(* Logix 5000 project; controller Proyecto_Final vendor 1 type 14 code 15 rev 16.42; software revision 16.03 *)

TASK MainTask (continuous, watchdog 500 ms) : MainProgram

MODULES
   Local : vendor 1 type 14 code 15 (SoftLogixController 2, rev 16.42)
END_MODULES

ADD_ON_INSTRUCTION Motorr   (* revision 1.0 *)
// Add On Motor
VAR_INPUT
   Cmd_Run : BOOL; {visible}   // Comando para acticar el motor en modo automatico
   Cmd_Stop : BOOL; {visible}   // Comando para detener el motor en modo automatico
   HMI_Run : BOOL;   // Comando para acticar el motor en modo manual
   HMI_Stop : BOOL;   // Comando para detener el motor en modo automatico
   Inp_Running : BOOL; {visible}   // Confirmacion de Falla del Motor
END_VAR
VAR_OUTPUT
   Sts_Running : BOOL; {visible}   // Estado activo del motor(salida fisica del PLC)
   Sts_RunFault : BOOL; {visible}   // Estado de falla del motor
END_VAR
VAR_INPUT
   Modo_Operacion : BOOL;
END_VAR
VAR
   Auto_Running : BOOL;
   Manu_Runnung : BOOL;
   TimerFault : TIMER := (PRE := 6000);
END_VAR

ROUTINE Logic   (* ladder *)
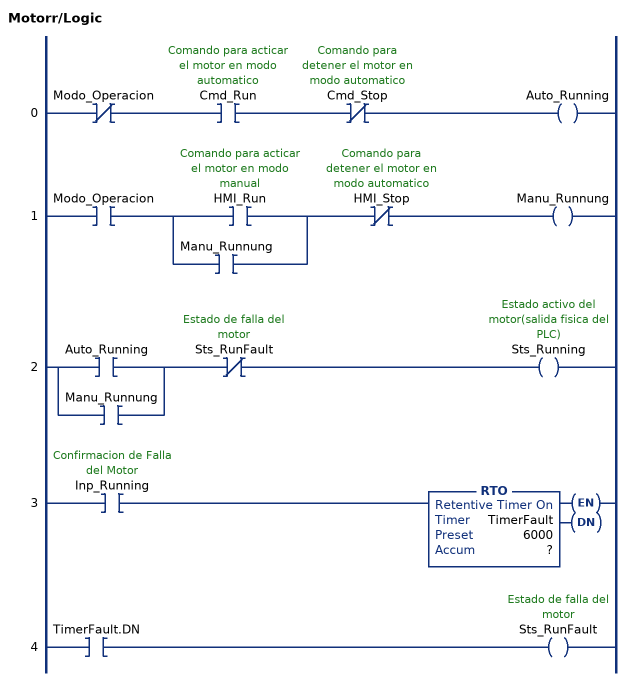
   0: XIO(Modo_Operacion)XIC(Cmd_Run)XIO(Cmd_Stop)OTE(Auto_Running);
   1: XIC(Modo_Operacion)[XIC(HMI_Run) ,XIC(Manu_Runnung) ]XIO(HMI_Stop)OTE(Manu_Runnung);
   2: [XIC(Auto_Running) ,XIC(Manu_Runnung) ]XIO(Sts_RunFault)OTE(Sts_Running);
   3: XIC(Inp_Running)RTO(TimerFault,?,?);
   4: XIC(TimerFault.DN)OTE(Sts_RunFault);
END_ROUTINE
END_ADD_ON_INSTRUCTION

ADD_ON_INSTRUCTION PICK_AND_PLACE   (* revision 1.0 *)
VAR_OUTPUT
   Banda_Entry_Conveyor : BOOL; {visible}
   Move_z : BOOL; {visible}
   Grab : BOOL; {visible}
   Move_x : BOOL; {visible}
   Banda_Exit_Conveyor : BOOL; {visible}
END_VAR
VAR_INPUT
   Sensor_Item_at_entry : BOOL;
   Sensor_Item_detected : BOOL;
   Sensor_Item_at_exit : BOOL;
   Cmd_Run_Banda_Entry_Conveyor : BOOL; {visible}
   Cmd_Run_Move_z : BOOL; {visible}
   Cmd_Run_Grab : BOOL; {visible}
   Cmd_Run_Move_x : BOOL; {visible}
   Cmd_Run_Banda_Exit_Conveyor : BOOL; {visible}
   Modo_Operacion : BOOL;
   Sensor_Entry : BOOL;
END_VAR

ROUTINE Logic   (* ladder *)
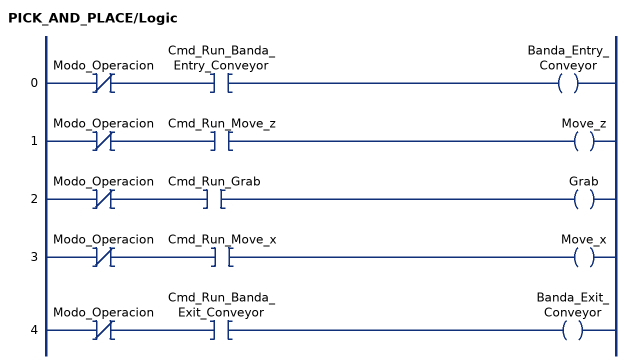
   0: XIO(Modo_Operacion)XIC(Cmd_Run_Banda_Entry_Conveyor)OTE(Banda_Entry_Conveyor);
   1: XIO(Modo_Operacion)XIC(Cmd_Run_Move_z)OTE(Move_z);
   2: XIO(Modo_Operacion)XIC(Cmd_Run_Grab)OTE(Grab);
   3: XIO(Modo_Operacion)XIC(Cmd_Run_Move_x)OTE(Move_x);
   4: XIO(Modo_Operacion)XIC(Cmd_Run_Banda_Exit_Conveyor)OTE(Banda_Exit_Conveyor);
END_ROUTINE
END_ADD_ON_INSTRUCTION

ADD_ON_INSTRUCTION PICK_AND_PLACE_XYZ   (* revision 1.0 *)
VAR_INPUT
   Modo_Operacion : BOOL; {visible}
   Cmd_Run_Pallet_Conveyor : BOOL; {visible}
   Cmd_Run_Part_Conveyor : BOOL; {visible}
   Cmd_Run_GradXYZ : BOOL; {visible}
END_VAR
VAR_OUTPUT
   Pallet_Conveyor : BOOL; {visible}
   Part_Conveyor : BOOL; {visible}
END_VAR
VAR_INPUT
   Sensor_Pallet : BOOL;
   Sensor_Part : BOOL;
   Sensor_Deteccion : BOOL;
END_VAR
VAR_OUTPUT
   V_Eje_X : REAL; {visible}
   V_Eje_Y : REAL; {visible}
   V_Eje_Z : REAL; {visible}
   GradXYZ : BOOL;
END_VAR
VAR_INPUT
   Sensor_Entry : BOOL;
   Cmd_Run_Emiter_Pallets : BOOL; {visible}
END_VAR
VAR_OUTPUT
   Emiter_Pallets : BOOL; {visible}
END_VAR

ROUTINE Logic   (* ladder *)
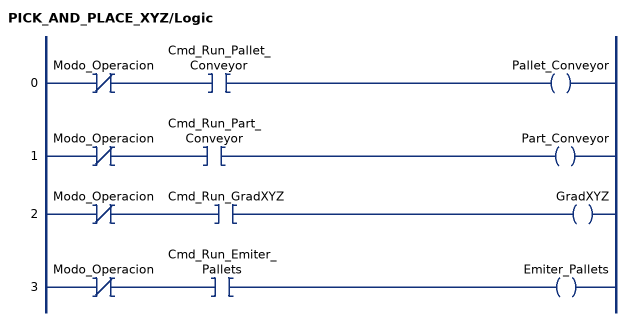
   0: XIO(Modo_Operacion)XIC(Cmd_Run_Pallet_Conveyor)OTE(Pallet_Conveyor);
   1: XIO(Modo_Operacion)XIC(Cmd_Run_Part_Conveyor)OTE(Part_Conveyor);
   2: XIO(Modo_Operacion)XIC(Cmd_Run_GradXYZ)OTE(GradXYZ);
   3: XIO(Modo_Operacion)XIC(Cmd_Run_Emiter_Pallets)OTE(Emiter_Pallets);
END_ROUTINE
END_ADD_ON_INSTRUCTION

ADD_ON_INSTRUCTION PRODUCTION_LINE   (* revision 1.0 *)
VAR_INPUT
   Modo_Operacion : BOOL; {visible}
   Cmd_Run_Banda_Lids_In : BOOL; {visible}
   Cmd_Run_Brazo : BOOL; {visible}
   Cmd_Run_Banda_Lids_Out1 : BOOL; {visible}
   Cmd_Run_Banda_Lids_Out2 : BOOL; {visible}
END_VAR
VAR_OUTPUT
   Banda_Lids_In : BOOL; {visible}
   Banda_Lids_Out1 : BOOL; {visible}
   Banda_Lids_Out2 : BOOL; {visible}
END_VAR
VAR_INPUT
   Sensor_Lid_In : BOOL;
   Sensor_Lid_Out : BOOL;
END_VAR
VAR_OUTPUT
   Brazo : BOOL; {visible}
END_VAR

ROUTINE Logic   (* ladder *)
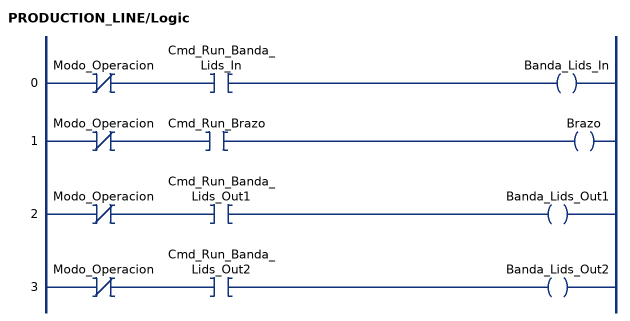
   0: XIO(Modo_Operacion)XIC(Cmd_Run_Banda_Lids_In)OTE(Banda_Lids_In);
   1: XIO(Modo_Operacion)XIC(Cmd_Run_Brazo)OTE(Brazo);
   2: XIO(Modo_Operacion)XIC(Cmd_Run_Banda_Lids_Out1)OTE(Banda_Lids_Out1);
   3: XIO(Modo_Operacion)XIC(Cmd_Run_Banda_Lids_Out2)OTE(Banda_Lids_Out2);
END_ROUTINE
END_ADD_ON_INSTRUCTION

ADD_ON_INSTRUCTION SCENE_1   (* revision 1.0 *)
VAR_INPUT
   Modo_Operacion : BOOL;   // Comando para cambiar el Modo_Automatico_Manual
   Item_at_entry : BOOL; {visible}
   Item_detected : BOOL; {visible}
   Item_at_exit : BOOL; {visible}
END_VAR
VAR_OUTPUT
   Entry_conveyor : BOOL; {visible}
   Move_z : BOOL; {visible}
   Grab : BOOL; {visible}
   Move_x : BOOL; {visible}
   Exit_coneyor : BOOL; {visible}
END_VAR
VAR_INPUT
   Incio : BOOL; {visible}
   Mover_Banda_1 : BOOL; {visible}
END_VAR
VAR_OUTPUT
   Banda_1 : BOOL; {visible}
END_VAR
VAR_INPUT
   Mover_eje_z : BOOL; {visible}
   Sostener_Pieza : BOOL; {visible}
   Mover_banda_2 : BOOL; {visible}
   Mover_eje_x : BOOL; {visible}
END_VAR
VAR
   Timer_Axis : TIMER := (PRE := 1000);
   Inicio : BOOL;
END_VAR

ROUTINE Logic   (* ladder *)
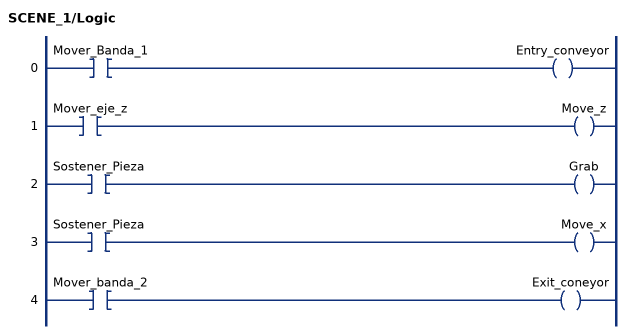
   0: XIC(Mover_Banda_1)OTE(Entry_conveyor);
   1: XIC(Mover_eje_z)OTE(Move_z);
   2: XIC(Sostener_Pieza)OTE(Grab);
   3: XIC(Sostener_Pieza)OTE(Move_x);
   4: XIC(Mover_banda_2)OTE(Exit_coneyor);
END_ROUTINE
END_ADD_ON_INSTRUCTION

ADD_ON_INSTRUCTION SEPARATION_STATION   (* revision 1.0 *)
VAR_INPUT
   Modo_Operacion : BOOL; {visible}
   Cmd_Run_Banda_Conveyor : BOOL; {visible}
   Cmd_Run_Pusher_Green : BOOL; {visible}
   Cmd_Run_Pusher_Blue : BOOL; {visible}
   Sensor_Piezas_Green : DINT; {visible}
   Sensor_Piezas_Blue : DINT; {visible}
END_VAR
VAR_OUTPUT
   Banda_Conveyor : BOOL; {visible}
   Pusher_Green : BOOL; {visible}
   Pusher_Bluee : BOOL; {visible}
END_VAR
VAR_INPUT
   Sensor_Entry : BOOL;
END_VAR

ROUTINE Logic   (* ladder *)
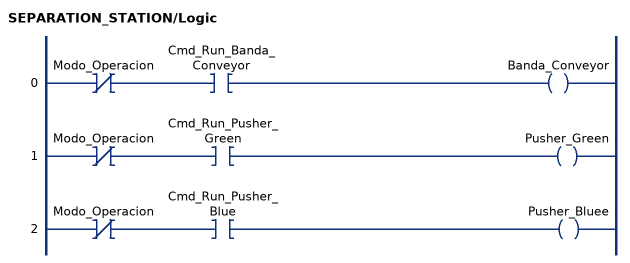
   0: XIO(Modo_Operacion)XIC(Cmd_Run_Banda_Conveyor)OTE(Banda_Conveyor);
   1: XIO(Modo_Operacion)XIC(Cmd_Run_Pusher_Green)OTE(Pusher_Green);
   2: XIO(Modo_Operacion)XIC(Cmd_Run_Pusher_Blue)OTE(Pusher_Bluee);
END_ROUTINE
END_ADD_ON_INSTRUCTION

ADD_ON_INSTRUCTION SORTING_BY_HEIGHT   (* revision 1.0 *)
VAR_INPUT
   Modo_Operacion : BOOL; {visible}
   Cmd_Run_Conveyor_Entry : BOOL; {visible}
   Cmd_Run_Load : BOOL; {visible}
   Cmd_Run_Turn : BOOL; {visible}
   Cmd_Run_Conveyor_Right : BOOL; {visible}
   Cmd_Run_Conveyor_Left : BOOL; {visible}
   Cmd_Run_Un_Load : BOOL; {visible}
END_VAR
VAR_OUTPUT
   Conveyor_Entry : BOOL; {visible}
   Load : BOOL; {visible}
   Turn : BOOL; {visible}
   Conveyor_Right : BOOL; {visible}
   Conveyor_Left : BOOL; {visible}
   Un_Load : BOOL; {visible}
END_VAR
VAR_INPUT
   Sensor_Low : BOOL;
   Sensor_High : BOOL;
   Sensor_Final_Conveyor_Entry : BOOL;
   Sensor_Front : BOOL;
   Sensor_In_Right_Conveyor : BOOL;
   Sensor_In_Left_Conveyor : BOOL;
   Sensor_Entry : BOOL;
END_VAR

ROUTINE Logic   (* ladder *)
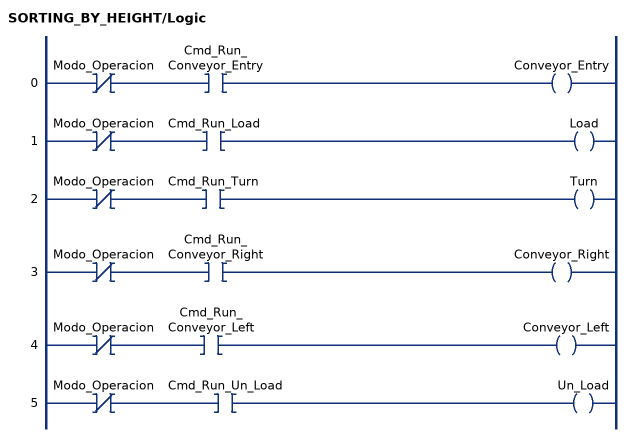
   0: XIO(Modo_Operacion)XIC(Cmd_Run_Conveyor_Entry)OTE(Conveyor_Entry);
   1: XIO(Modo_Operacion)XIC(Cmd_Run_Load)OTE(Load);
   2: XIO(Modo_Operacion)XIC(Cmd_Run_Turn)OTE(Turn);
   3: XIO(Modo_Operacion)XIC(Cmd_Run_Conveyor_Right)OTE(Conveyor_Right);
   4: XIO(Modo_Operacion)XIC(Cmd_Run_Conveyor_Left)OTE(Conveyor_Left);
   5: XIO(Modo_Operacion)XIC(Cmd_Run_Un_Load)OTE(Un_Load);
END_ROUTINE
END_ADD_ON_INSTRUCTION

ADD_ON_INSTRUCTION SORTING_BY_WEIGHT   (* revision 1.0 *)
VAR_INPUT
   Modo_Operacion : BOOL; {visible}
   Cmd_Run_Conveyor_Entry : BOOL; {visible}
   Cmd_Run_Conveyor_Peso : BOOL; {visible}
   Cmd_Run_Send_Adelante : BOOL; {visible}
   Cmd_Run_Send_Right : BOOL; {visible}
   Cmd_Run_Send_Left : BOOL; {visible}
   Cmd_Run_Conveyor_Right : BOOL; {visible}
   Cmd_Run_Conveyor_Left : BOOL; {visible}
   Cmd_Run_Conveyor_Front : BOOL; {visible}
END_VAR
VAR_OUTPUT
   Conveyor_Entry : BOOL; {visible}
   Conveyor_Peso : BOOL; {visible}
   Send_Adelante : BOOL; {visible}
   Send_Right : BOOL; {visible}
   Send_Left : BOOL; {visible}
   Conveyor_Right : BOOL; {visible}
   Conveyor_Left : BOOL; {visible}
   Conveyor_Front : BOOL; {visible}
END_VAR
VAR_INPUT
   Sensor_Peso : REAL; {visible}
   Sensor_Conveyor_Entry : BOOL;
   Sensor_Conveyor_In_Right : BOOL;
   Sensor_Conveyor_In_Left : BOOL;
   Sensor_Conveyor_In_Front : BOOL;
END_VAR

ROUTINE Logic   (* ladder *)
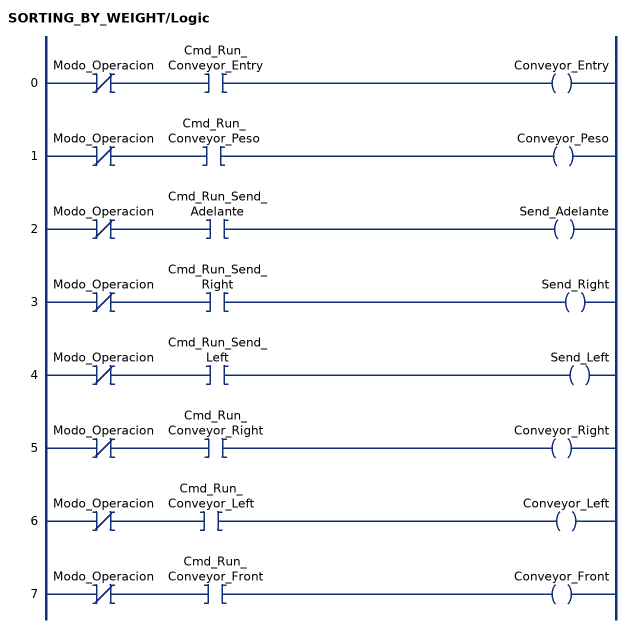
   0: XIO(Modo_Operacion)XIC(Cmd_Run_Conveyor_Entry)OTE(Conveyor_Entry);
   1: XIO(Modo_Operacion)XIC(Cmd_Run_Conveyor_Peso)OTE(Conveyor_Peso);
   2: XIO(Modo_Operacion)XIC(Cmd_Run_Send_Adelante)OTE(Send_Adelante);
   3: XIO(Modo_Operacion)XIC(Cmd_Run_Send_Right)OTE(Send_Right);
   4: XIO(Modo_Operacion)XIC(Cmd_Run_Send_Left)OTE(Send_Left);
   5: XIO(Modo_Operacion)XIC(Cmd_Run_Conveyor_Right)OTE(Conveyor_Right);
   6: XIO(Modo_Operacion)XIC(Cmd_Run_Conveyor_Left)OTE(Conveyor_Left);
   7: XIO(Modo_Operacion)XIC(Cmd_Run_Conveyor_Front)OTE(Conveyor_Front);
END_ROUTINE
END_ADD_ON_INSTRUCTION

VAR_GLOBAL   (* controller tags *)
   A1 : SFC_STEP;
   AAAA : SFC_STEP;
   Altura : SORTING_BY_HEIGHT;
   AZU : BOOL;
   B1 : SFC_STEP;
   BBB : SFC_STEP;
   BBB_001 : SFC_STEP;
   BBB_002 : SFC_STEP;
   BBB_003 : SFC_STEP;
   BOOL_IN_0 : ALIAS FOR Proceso.Sensor_Item_at_entry;
   BOOL_IN_1 : ALIAS FOR Proceso.Sensor_Item_detected;
   BOOL_IN_10 : ALIAS FOR Proceso2.Sensor_Entry;
   BOOL_IN_11 : ALIAS FOR STARTR;
   BOOL_IN_12 : ALIAS FOR Linea1.Sensor_Lid_In;
   BOOL_IN_13 : ALIAS FOR Linea1.Sensor_Lid_Out;
   BOOL_IN_14 : ALIAS FOR Linea2.Sensor_Lid_In;
   BOOL_IN_15 : ALIAS FOR Linea2.Sensor_Lid_Out;
   BOOL_IN_16 : ALIAS FOR Proceso.Sensor_Entry;
   BOOL_IN_17 : ALIAS FOR XYZ.Sensor_Pallet;
   BOOL_IN_18 : ALIAS FOR XYZ.Sensor_Part;
   BOOL_IN_19 : ALIAS FOR XYZ.Sensor_Deteccion;
   BOOL_IN_2 : ALIAS FOR Proceso.Sensor_Item_at_exit;
   BOOL_IN_20 : ALIAS FOR SEPARA.Sensor_Entry;
   BOOL_IN_21 : ALIAS FOR Altura.Sensor_Low;
   BOOL_IN_22 : ALIAS FOR Altura.Sensor_Final_Conveyor_Entry;
   BOOL_IN_23 : ALIAS FOR Altura.Sensor_Front;
   BOOL_IN_24 : ALIAS FOR Altura.Sensor_In_Right_Conveyor;
   BOOL_IN_25 : ALIAS FOR Altura.Sensor_High;
   BOOL_IN_26 : ALIAS FOR Altura.Sensor_In_Left_Conveyor;
   BOOL_IN_27 : ALIAS FOR Peso.Sensor_Conveyor_Entry;
   BOOL_IN_28 : ALIAS FOR Peso.Sensor_Conveyor_In_Right;
   BOOL_IN_29 : ALIAS FOR Peso.Sensor_Conveyor_In_Left;
   BOOL_IN_3 : ALIAS FOR Line3.Sensor_Lid_In;
   BOOL_IN_30 : ALIAS FOR Peso.Sensor_Conveyor_In_Front;
   BOOL_IN_31 : ALIAS FOR REARME;
   BOOL_IN_32 : ALIAS FOR STOPSITO;
   BOOL_IN_4 : ALIAS FOR Line3.Sensor_Lid_Out;
   BOOL_IN_5 : ALIAS FOR XYZ.Sensor_Entry;
   BOOL_IN_6 : ALIAS FOR Altura.Sensor_Entry;
   BOOL_IN_7 : ALIAS FOR Proceso2.Sensor_Item_at_entry;
   BOOL_IN_8 : ALIAS FOR Proceso2.Sensor_Item_detected;
   BOOL_IN_9 : ALIAS FOR Proceso2.Sensor_Item_at_exit;
   BOOL_OUT_0 : ALIAS FOR Proceso.Banda_Entry_Conveyor;
   BOOL_OUT_1 : ALIAS FOR Proceso.Move_z;
   BOOL_OUT_10 : ALIAS FOR Line3.Banda_Lids_Out1;
   BOOL_OUT_11 : ALIAS FOR Line3.Banda_Lids_Out2;
   BOOL_OUT_12 : ALIAS FOR Linea1.Banda_Lids_In;
   BOOL_OUT_13 : ALIAS FOR Linea1.Brazo;
   BOOL_OUT_14 : ALIAS FOR Linea1.Banda_Lids_Out1;
   BOOL_OUT_15 : ALIAS FOR Linea1.Banda_Lids_Out2;
   BOOL_OUT_16 : ALIAS FOR Linea2.Banda_Lids_In;
   BOOL_OUT_17 : ALIAS FOR Linea2.Brazo;
   BOOL_OUT_18 : ALIAS FOR Linea2.Banda_Lids_Out1;
   BOOL_OUT_19 : ALIAS FOR Linea2.Banda_Lids_Out2;
   BOOL_OUT_2 : ALIAS FOR Proceso.Grab;
   BOOL_OUT_20 : ALIAS FOR XYZ.Pallet_Conveyor;
   BOOL_OUT_21 : ALIAS FOR XYZ.Part_Conveyor;
   BOOL_OUT_22 : ALIAS FOR XYZ.GradXYZ;
   BOOL_OUT_23 : ALIAS FOR Altura.Conveyor_Entry;
   BOOL_OUT_24 : ALIAS FOR Altura.Load;
   BOOL_OUT_25 : ALIAS FOR Altura.Turn;
   BOOL_OUT_26 : ALIAS FOR Altura.Conveyor_Right;
   BOOL_OUT_27 : ALIAS FOR Altura.Un_Load;
   BOOL_OUT_28 : ALIAS FOR Altura.Conveyor_Left;
   BOOL_OUT_29 : ALIAS FOR Peso.Conveyor_Entry;
   BOOL_OUT_3 : ALIAS FOR Proceso.Move_x;
   BOOL_OUT_30 : ALIAS FOR Peso.Conveyor_Peso;
   BOOL_OUT_31 : ALIAS FOR Peso.Send_Right;
   BOOL_OUT_32 : ALIAS FOR Peso.Send_Adelante;
   BOOL_OUT_33 : ALIAS FOR Peso.Conveyor_Right;
   BOOL_OUT_34 : ALIAS FOR Peso.Send_Left;
   BOOL_OUT_35 : ALIAS FOR Peso.Conveyor_Left;
   BOOL_OUT_36 : ALIAS FOR Peso.Conveyor_Front;
   BOOL_OUT_37 : ALIAS FOR XYZ.Emiter_Pallets;
   BOOL_OUT_39 : ALIAS FOR Proceso2.Move_z;
   BOOL_OUT_4 : ALIAS FOR Proceso.Banda_Exit_Conveyor;
   BOOL_OUT_40 : ALIAS FOR Proceso2.Grab;
   BOOL_OUT_41 : ALIAS FOR Proceso2.Move_x;
   BOOL_OUT_42 : ALIAS FOR Proceso2.Banda_Entry_Conveyor;
   BOOL_OUT_43 : ALIAS FOR Proceso2.Banda_Exit_Conveyor;
   BOOL_OUT_5 : ALIAS FOR SEPARA.Banda_Conveyor;
   BOOL_OUT_6 : ALIAS FOR SEPARA.Pusher_Green;
   BOOL_OUT_7 : ALIAS FOR SEPARA.Pusher_Bluee;
   BOOL_OUT_8 : ALIAS FOR Line3.Banda_Lids_In;
   BOOL_OUT_9 : ALIAS FOR Line3.Brazo;
   C1 : SFC_STEP;
   CC : SFC_STEP;
   CC_001 : SFC_STEP;
   CC_002 : SFC_STEP;
   CC_003 : SFC_STEP;
   CMD_1 : BOOL;
   CMD_2 : BOOL;
   CMD_3 : BOOL;
   Cmd_banda1 : BOOL;
   Cmd_banda2 : BOOL;
   Cmd_banda3 : BOOL;
   CMD_banda_derecha : BOOL;
   CMD_banda_Front : BOOL;
   CMD_banda_IZQQ : BOOL;
   Cmd_bandaCLAS : BOOL;
   CMD_conveyor_entry : BOOL;
   CMD_conveyor_peso : BOOL;
   CMD_DETEC : BOOL;
   Cmd_giro : BOOL;
   CMD_LEFT : BOOL;
   Cmd_LOAD : BOOL;
   CMD_RIFHT : BOOL;
   CMD_Send_Front : BOOL;
   CMD_Send_LEFT : BOOL;
   CMD_Send_righ : BOOL;
   CMD_Send_ruedas : BOOL;
   Cmd_Turn : BOOL;
   CMD_UNLOAD : BOOL;
   CMD_X : BOOL;
   CMD_X0 : BOOL;
   CMD_X2 : BOOL;
   CMD_Y : BOOL;
   CMD_Y0 : BOOL;
   CMD_Y2 : BOOL;
   CMD_Z : BOOL;
   CMD_Z0 : BOOL;
   CMD_Z2 : BOOL;
   CMDGIRO : BOOL;
   D1 : SFC_STEP;
   DD : SFC_STEP;
   DD_001 : SFC_STEP;
   DD_002 : SFC_STEP;
   DD_003 : SFC_STEP;
   DF : SFC_STEP := (PRE := 100);
   DF_001 : SFC_STEP := (PRE := 100);
   DF_002 : SFC_STEP := (PRE := 100);
   DFR : SFC_STEP := (PRE := 4000);
   E1 : SFC_STEP := (PRE := 2500);
   E1_001 : SFC_STEP := (PRE := 2500);
   E1_002 : SFC_STEP := (PRE := 2500);
   E2 : SFC_STEP;
   E2_001 : SFC_STEP;
   E2_002 : SFC_STEP;
   E3 : SFC_STEP := (PRE := 1200);
   E3_001 : SFC_STEP := (PRE := 1200);
   E3_002 : SFC_STEP := (PRE := 1200);
   E3_003 : SFC_STEP := (PRE := 1200);
   E3_004 : SFC_STEP := (PRE := 1200);
   E3_005 : SFC_STEP := (PRE := 1200);
   E3_006 : SFC_STEP := (PRE := 1200);
   E3_007 : SFC_STEP := (PRE := 1200);
   E4 : SFC_STEP := (PRE := 600);
   E4_001 : SFC_STEP := (PRE := 600);
   E4_002 : SFC_STEP := (PRE := 600);
   E4_003 : SFC_STEP := (PRE := 425);
   E4_004 : SFC_STEP := (PRE := 600);
   E4_005 : SFC_STEP := (PRE := 425);
   E4_006 : SFC_STEP := (PRE := 350);
   E4_007 : SFC_STEP := (PRE := 600);
   EE : SFC_STEP := (PRE := 350);
   EE_001 : SFC_STEP := (PRE := 350);
   EE_002 : SFC_STEP := (PRE := 350);
   EE_003 : SFC_STEP := (PRE := 350);
   EO : DINT;
   EOwww : SFC_STEP;
   EOwww_001 : SFC_STEP;
   ERT : SFC_STEP;
   ERTT : SFC_STEP;
   ERTT_001 : SFC_STEP;
   ERTT_002 : SFC_STEP;
   ET1 : SFC_STEP;
   ET10 : SFC_STEP := (PRE := 1200);
   ET11 : SFC_STEP := (PRE := 1200);
   ET12 : SFC_STEP;
   ET122 : SFC_STEP;
   ET3 : SFC_STEP;
   ET4 : SFC_STEP;
   ET4_001 : SFC_STEP;
   ET5 : SFC_STEP;
   ET5_001 : SFC_STEP;
   ET6 : SFC_STEP;
   ET7 : SFC_STEP;
   ET8 : SFC_STEP;
   ET89 : SFC_STEP;
   ET9 : SFC_STEP := (PRE := 1200);
   ETP1 : SFC_STEP;
   ETP2 : SFC_STEP;
   ETP22 : SFC_STEP := (PRE := 2500);
   ETP3 : SFC_STEP;
   ETP4 : SFC_STEP := (PRE := 1200);
   ETP5 : SFC_STEP := (PRE := 600);
   ETP6 : SFC_STEP := (PRE := 4000);
   ETP66 : SFC_STEP := (PRE := 2700);
   ETY1 : SFC_STEP := (PRE := 4000);
   ETY1_001 : SFC_STEP := (PRE := 4000);
   EYT : SFC_STEP;
   F1 : SFC_STEP := (PRE := 3000);
   F1_001 : SFC_STEP := (PRE := 3000);
   FF : SFC_STEP := (PRE := 1000);
   FF_001 : SFC_STEP := (PRE := 1000);
   FF_002 : SFC_STEP := (PRE := 1000);
   FF_003 : SFC_STEP := (PRE := 1000);
   FG : SFC_STEP;
   FG_001 : SFC_STEP;
   FG_002 : SFC_STEP;
   FLOAT_IN_0 : REAL;
   FLOAT_IN_1 : DINT;
   FLOAT_IN_2 : REAL;
   FLOAT_IN_3 : ALIAS FOR Peso.Sensor_Peso;
   FLOAT_IN_ON : DINT;
   FLOAT_OUT_0 : ALIAS FOR XYZ.V_Eje_X;
   FLOAT_OUT_1 : ALIAS FOR XYZ.V_Eje_Y;
   FLOAT_OUT_2 : ALIAS FOR XYZ.V_Eje_Z;
   G1 : SFC_STEP;
   GGG : SFC_STEP := (PRE := 150);
   GGG_001 : SFC_STEP := (PRE := 150);
   GGG_002 : SFC_STEP := (PRE := 150);
   GGG_003 : SFC_STEP := (PRE := 150);
   III : SFC_STEP;
   INT_IN_0 : ALIAS FOR SEPARA.Sensor_Piezas_Blue;
   INT_IN_1 : ALIAS FOR SEPARA.Sensor_Piezas_Green;
   INT_OUT_0 : REAL;
   INT_OUT_1 : DINT;
   INT_OUT_O : DINT;
   IO : SFC_STEP;
   IO_001 : SFC_STEP;
   IO_002 : SFC_STEP;
   KKK : SFC_STEP := (PRE := 7000);
   KKK_001 : SFC_STEP := (PRE := 4000);
   Line3 : PRODUCTION_LINE;
   Linea1 : PRODUCTION_LINE;
   Linea2 : PRODUCTION_LINE;
   Modo_Operacion : BOOL;
   Peso : SORTING_BY_WEIGHT;
   Proceso : PICK_AND_PLACE;
   Proceso1 : BOOL;
   Proceso2 : PICK_AND_PLACE;
   prueba : TIMER := (PRE := 6);
   QW : SFC_STEP;
   RE : SFC_STEP := (PRE := 330);
   RE_001 : SFC_STEP := (PRE := 330);
   RE_002 : SFC_STEP := (PRE := 330);
   REARME : BOOL;
   REPIT : SFC_STEP;
   RRR : SFC_STEP;
   RRR_001 : SFC_STEP;
   RRR_002 : SFC_STEP;
   RT : SFC_STEP;
   RT_001 : SFC_STEP;
   RT_002 : SFC_STEP;
   SEPARA : SEPARATION_STATION;
   START1 : BOOL;
   STARTR : BOOL;
   STARTT : BOOL;
   STOP2 : BOOL;
   STOPSITO : BOOL;
   SYS_0N : BOOL;
   T2 : SFC_STEP;
   T2_001 : SFC_STEP;
   T2_002 : SFC_STEP;
   test : BOOL;
   TESTTT : TIMER := (PRE := 6);
   testttt : TIMER := (PRE := 5000);
   tiempo : BOOL;
   TR : SFC_STEP;
   TR_001 : SFC_STEP;
   TR_002 : SFC_STEP;
   TTT : BOOL;
   ty : SFC_STEP := (Count := 2);
   V1 : SFC_STEP := (PRE := 3000);
   VER : BOOL;
   WE : SFC_STEP;
   WEE : SFC_STEP := (PRE := 1000);
   WEE_001 : SFC_STEP := (PRE := 1000);
   WERR : SFC_STEP;
   X1 : SFC_STEP;
   XX : SFC_STEP;
   XX_001 : SFC_STEP;
   XX_002 : SFC_STEP;
   XYZ : PICK_AND_PLACE_XYZ;
   Y1 : SFC_STEP := (PRE := 2500);
   Z1 : SFC_STEP;
END_VAR

PROGRAM MainProgram   (* main routine MainRoutine *)
VAR
   Action_000 : SFC_ACTION;
   Action_001 : SFC_ACTION;
   Action_002 : SFC_ACTION;
   Action_003 : SFC_ACTION;
   Action_004 : SFC_ACTION;
   Action_005 : SFC_ACTION;
   Action_006 : SFC_ACTION;
   Action_007 : SFC_ACTION;
   Action_008 : SFC_ACTION;
   Action_009 : SFC_ACTION;
   Action_010 : SFC_ACTION;
   Action_011 : SFC_ACTION;
   Action_012 : SFC_ACTION;
   Action_013 : SFC_ACTION;
   Action_014 : SFC_ACTION;
   Action_015 : SFC_ACTION;
   Action_016 : SFC_ACTION;
   Action_017 : SFC_ACTION;
   Action_018 : SFC_ACTION;
   Action_019 : SFC_ACTION;
   Action_020 : SFC_ACTION;
   Action_021 : SFC_ACTION;
   Action_022 : SFC_ACTION;
   Action_023 : SFC_ACTION;
   Action_024 : SFC_ACTION;
   Action_025 : SFC_ACTION;
   Action_026 : SFC_ACTION;
   Action_027 : SFC_ACTION;
   Action_028 : SFC_ACTION;
   Action_029 : SFC_ACTION;
   Action_030 : SFC_ACTION;
   Action_031 : SFC_ACTION;
   Action_032 : SFC_ACTION;
   Action_033 : SFC_ACTION;
   Action_034 : SFC_ACTION;
   Action_035 : SFC_ACTION;
   Action_036 : SFC_ACTION;
   Action_037 : SFC_ACTION;
   Action_038 : SFC_ACTION;
   Action_039 : SFC_ACTION;
   Action_040 : SFC_ACTION;
   Action_041 : SFC_ACTION;
   Action_042 : SFC_ACTION;
   Action_043 : SFC_ACTION;
   Action_044 : SFC_ACTION;
   Action_045 : SFC_ACTION;
   Action_046 : SFC_ACTION;
   Action_047 : SFC_ACTION;
   Action_048 : SFC_ACTION;
   Action_049 : SFC_ACTION;
   Action_050 : SFC_ACTION;
   Action_051 : SFC_ACTION;
   Action_052 : SFC_ACTION;
   Action_053 : SFC_ACTION;
   Action_054 : SFC_ACTION;
   Action_055 : SFC_ACTION;
   Action_056 : SFC_ACTION;
   Action_057 : SFC_ACTION;
   Action_058 : SFC_ACTION;
   Action_059 : SFC_ACTION;
   Action_060 : SFC_ACTION;
   Action_061 : SFC_ACTION;
   Action_062 : SFC_ACTION;
   Action_063 : SFC_ACTION;
   Action_064 : SFC_ACTION;
   Action_065 : SFC_ACTION;
   Action_066 : SFC_ACTION;
   Action_067 : SFC_ACTION;
   Action_068 : SFC_ACTION;
   Action_069 : SFC_ACTION;
   Action_070 : SFC_ACTION;
   Action_071 : SFC_ACTION;
   Action_072 : SFC_ACTION;
   Action_073 : SFC_ACTION;
   Action_074 : SFC_ACTION;
   Action_075 : SFC_ACTION;
   Action_076 : SFC_ACTION;
   Action_077 : SFC_ACTION;
   Action_078 : SFC_ACTION;
   Action_079 : SFC_ACTION;
   Action_080 : SFC_ACTION;
   Action_081 : SFC_ACTION;
   Action_082 : SFC_ACTION;
   Action_083 : SFC_ACTION;
   Action_084 : SFC_ACTION;
   Action_085 : SFC_ACTION;
   Action_086 : SFC_ACTION;
   Action_087 : SFC_ACTION;
   Action_088 : SFC_ACTION;
   Action_089 : SFC_ACTION;
   Action_090 : SFC_ACTION;
   Action_091 : SFC_ACTION;
   Action_092 : SFC_ACTION;
   Action_093 : SFC_ACTION;
   Action_094 : SFC_ACTION;
   Action_095 : SFC_ACTION;
   Action_096 : SFC_ACTION;
   Action_097 : SFC_ACTION;
   Action_098 : SFC_ACTION;
   ESCENA_1_01 : PICK_AND_PLACE;
   HIGH : DINT;
   Linea3 : PRODUCTION_LINE;
   Motorr_01 : Motorr;
   PICK_AND_PLACE_01 : PICK_AND_PLACE;
   PICK_AND_PLACE_XYZ_01 : PICK_AND_PLACE_XYZ;
   PRODUCTION_LINE_01 : PRODUCTION_LINE;
   SCENE_1_01 : SCENE_1;
   SEPARATIN_STATION_01 : SEPARATION_STATION;
   SORTING_BY_HEIGHT_01 : SORTING_BY_HEIGHT;
   SORTING_BY_WEIGHT_01 : SORTING_BY_WEIGHT;
   Step_000 : SFC_STEP;
   Step_001 : SFC_STEP;
   Step_002 : SFC_STEP;
   Step_003 : SFC_STEP;
   Step_004 : SFC_STEP;
   Step_005 : SFC_STEP;
   Step_006 : SFC_STEP;
   Step_007 : SFC_STEP;
   Step_008 : SFC_STEP;
   Step_009 : SFC_STEP;
   Step_010 : SFC_STEP;
   Step_011 : SFC_STEP;
   Step_012 : SFC_STEP;
   Step_013 : SFC_STEP := (PRE := 850);
   Step_014 : SFC_STEP := (PRE := 1000);
   Step_015 : SFC_STEP := (PRE := 1000);
   Step_016 : SFC_STEP := (PRE := 850);
   Step_017 : SFC_STEP;
   Step_018 : SFC_STEP;
   Step_019 : SFC_STEP;
   Step_020 : SFC_STEP;
   Step_021 : SFC_STEP;
   Step_022 : SFC_STEP;
   Step_023 : SFC_STEP;
   Step_024 : SFC_STEP;
   Step_025 : SFC_STEP;
   Step_026 : SFC_STEP;
   Step_027 : SFC_STEP;
   Step_028 : SFC_STEP;
   Step_029 : SFC_STEP;
   Step_030 : SFC_STEP;
   Step_031 : SFC_STEP;
   Step_032 : SFC_STEP;
   Step_033 : SFC_STEP;
   Step_034 : SFC_STEP;
   Step_035 : SFC_STEP;
   Step_036 : SFC_STEP;
   Step_037 : SFC_STEP;
   Step_038 : SFC_STEP;
   Step_039 : SFC_STEP;
   Step_040 : SFC_STEP;
   Step_041 : SFC_STEP;
   Step_042 : SFC_STEP;
   Step_043 : SFC_STEP;
   Step_044 : SFC_STEP;
   Step_045 : SFC_STEP;
   Step_046 : SFC_STEP;
   Step_047 : SFC_STEP;
   Step_048 : SFC_STEP;
   Step_049 : SFC_STEP;
   Step_050 : SFC_STEP;
   Step_051 : SFC_STEP := (PRE := 5000);
   Step_052 : SFC_STEP;
   Step_053 : SFC_STEP;
   Step_054 : SFC_STEP;
   Step_055 : SFC_STEP;
   Step_056 : SFC_STEP;
   Step_057 : SFC_STEP;
   Step_058 : SFC_STEP;
   Step_059 : SFC_STEP;
   Step_060 : SFC_STEP;
   Step_061 : SFC_STEP;
   Step_062 : SFC_STEP;
   Step_063 : SFC_STEP;
   Step_064 : SFC_STEP := (PRE := 1200);
   Step_065 : SFC_STEP;
   Step_066 : SFC_STEP;
   Step_067 : SFC_STEP;
   Step_068 : SFC_STEP;
   Tran_000 : BOOL;
   Tran_001 : BOOL;
   Tran_002 : BOOL;
   Tran_003 : BOOL;
   Tran_004 : BOOL;
   Tran_005 : BOOL;
   Tran_006 : BOOL;
   Tran_007 : BOOL;
   Tran_008 : BOOL;
   Tran_009 : BOOL;
   Tran_010 : BOOL;
   Tran_011 : BOOL;
   Tran_012 : BOOL;
   Tran_013 : BOOL;
   Tran_014 : BOOL;
   Tran_015 : BOOL;
   Tran_016 : BOOL;
   Tran_017 : BOOL;
   Tran_018 : BOOL;
   Tran_019 : BOOL;
   Tran_020 : BOOL;
   Tran_021 : BOOL;
   Tran_022 : BOOL;
   Tran_023 : BOOL;
   Tran_024 : BOOL;
   Tran_025 : BOOL;
   Tran_026 : BOOL;
   Tran_027 : BOOL;
   Tran_028 : BOOL;
   Tran_029 : BOOL;
   Tran_030 : BOOL;
   Tran_031 : BOOL;
   Tran_032 : BOOL;
   Tran_033 : BOOL;
   Tran_034 : BOOL;
   Tran_035 : BOOL;
   Tran_036 : BOOL;
   Tran_037 : BOOL;
   Tran_038 : BOOL;
   Tran_039 : BOOL;
   Tran_040 : BOOL;
   Tran_041 : BOOL;
   Tran_042 : BOOL;
   Tran_043 : BOOL;
   Tran_044 : BOOL;
   Tran_045 : BOOL;
   Tran_046 : BOOL;
   Tran_047 : BOOL;
   Tran_048 : BOOL;
   Tran_049 : BOOL;
   Tran_050 : BOOL;
   Tran_051 : BOOL;
   Tran_052 : BOOL;
   Tran_053 : BOOL;
   Tran_054 : BOOL;
   Tran_055 : BOOL;
   Tran_056 : BOOL;
   Tran_057 : BOOL;
   Tran_058 : BOOL;
   Tran_059 : BOOL;
   Tran_060 : BOOL;
   Tran_061 : BOOL;
   Tran_062 : BOOL;
   Tran_063 : BOOL;
   Tran_064 : BOOL;
   Tran_065 : BOOL;
   Tran_066 : BOOL;
   Tran_067 : BOOL;
   Tran_068 : BOOL;
   Tran_069 : BOOL;
   Tran_070 : BOOL;
   Tran_071 : BOOL;
   Tran_072 : BOOL;
   Tran_073 : BOOL;
   Tran_074 : BOOL;
   Tran_075 : BOOL;
   Tran_076 : BOOL;
   Tran_077 : BOOL;
   Tran_078 : BOOL;
   Tran_079 : BOOL;
   Tran_080 : BOOL;
   Tran_081 : BOOL;
   Tran_082 : BOOL;
   Tran_083 : BOOL;
   Tran_084 : BOOL;
   Tran_085 : BOOL;
   Tran_086 : BOOL;
   Tran_087 : BOOL;
   Tran_088 : BOOL;
   Tran_089 : BOOL;
   Tran_090 : BOOL;
   Tran_091 : BOOL;
   Tran_092 : BOOL;
   Tran_093 : BOOL;
   Tran_094 : BOOL;
   Tran_095 : BOOL;
   Tran_096 : BOOL;
   Tran_097 : BOOL;
   Tran_098 : BOOL;
   Tran_099 : BOOL;
   Tran_100 : BOOL;
   Tran_101 : BOOL;
   Tran_102 : BOOL;
   Tran_103 : BOOL;
   Tran_104 : BOOL;
   Tran_105 : BOOL;
   Tran_106 : BOOL;
   Tran_107 : BOOL;
   Tran_108 : BOOL;
   Tran_109 : BOOL;
   Tran_110 : BOOL;
   Tran_111 : BOOL;
   Tran_112 : BOOL;
   Tran_113 : BOOL;
   Tran_114 : BOOL;
   Tran_115 : BOOL;
   Tran_116 : BOOL;
   Tran_117 : BOOL;
   Tran_118 : BOOL;
END_VAR

ROUTINE equipos   (* function block diagram *)
   SHEET 1
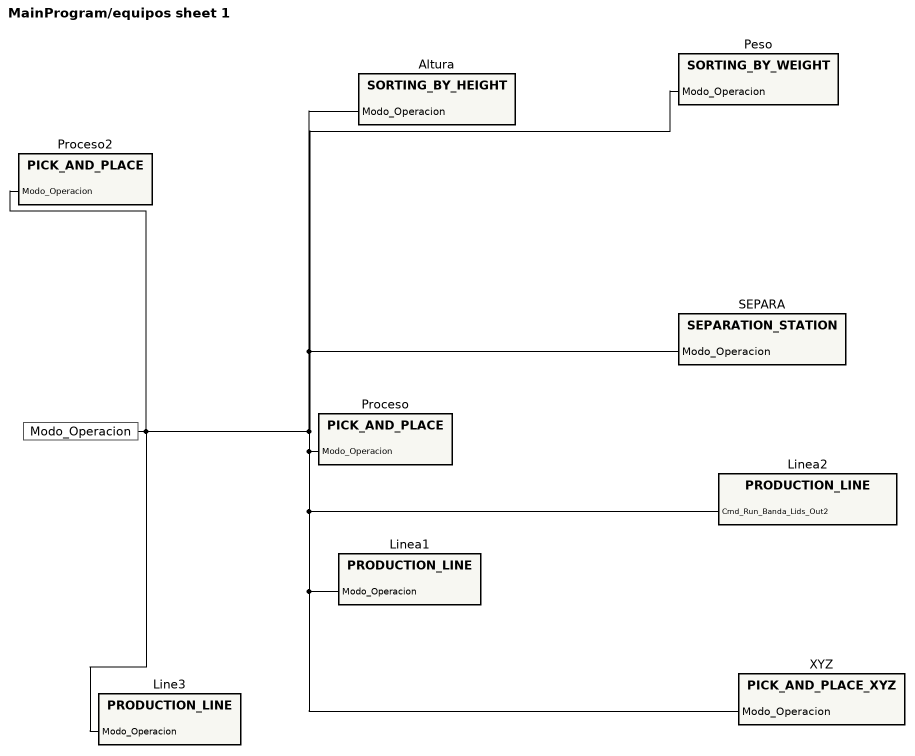
   Proceso2 : PICK_AND_PLACE(Modo_Operacion := Modo_Operacion);
   Line3 : PRODUCTION_LINE(Modo_Operacion := Modo_Operacion);
   Proceso : PICK_AND_PLACE(Modo_Operacion := Modo_Operacion);
   Linea1 : PRODUCTION_LINE(Modo_Operacion := Modo_Operacion);
   Altura : SORTING_BY_HEIGHT(Modo_Operacion := Modo_Operacion);
   Peso : SORTING_BY_WEIGHT(Modo_Operacion := Modo_Operacion);
   SEPARA : SEPARATION_STATION(Modo_Operacion := Modo_Operacion);
   Linea2 : PRODUCTION_LINE(Cmd_Run_Banda_Lids_Out2 := Modo_Operacion);
   XYZ : PICK_AND_PLACE_XYZ(Modo_Operacion := Modo_Operacion);
END_ROUTINE

ROUTINE ESCEN_1_PICK_AND_PLACE   (* sequential function chart *)
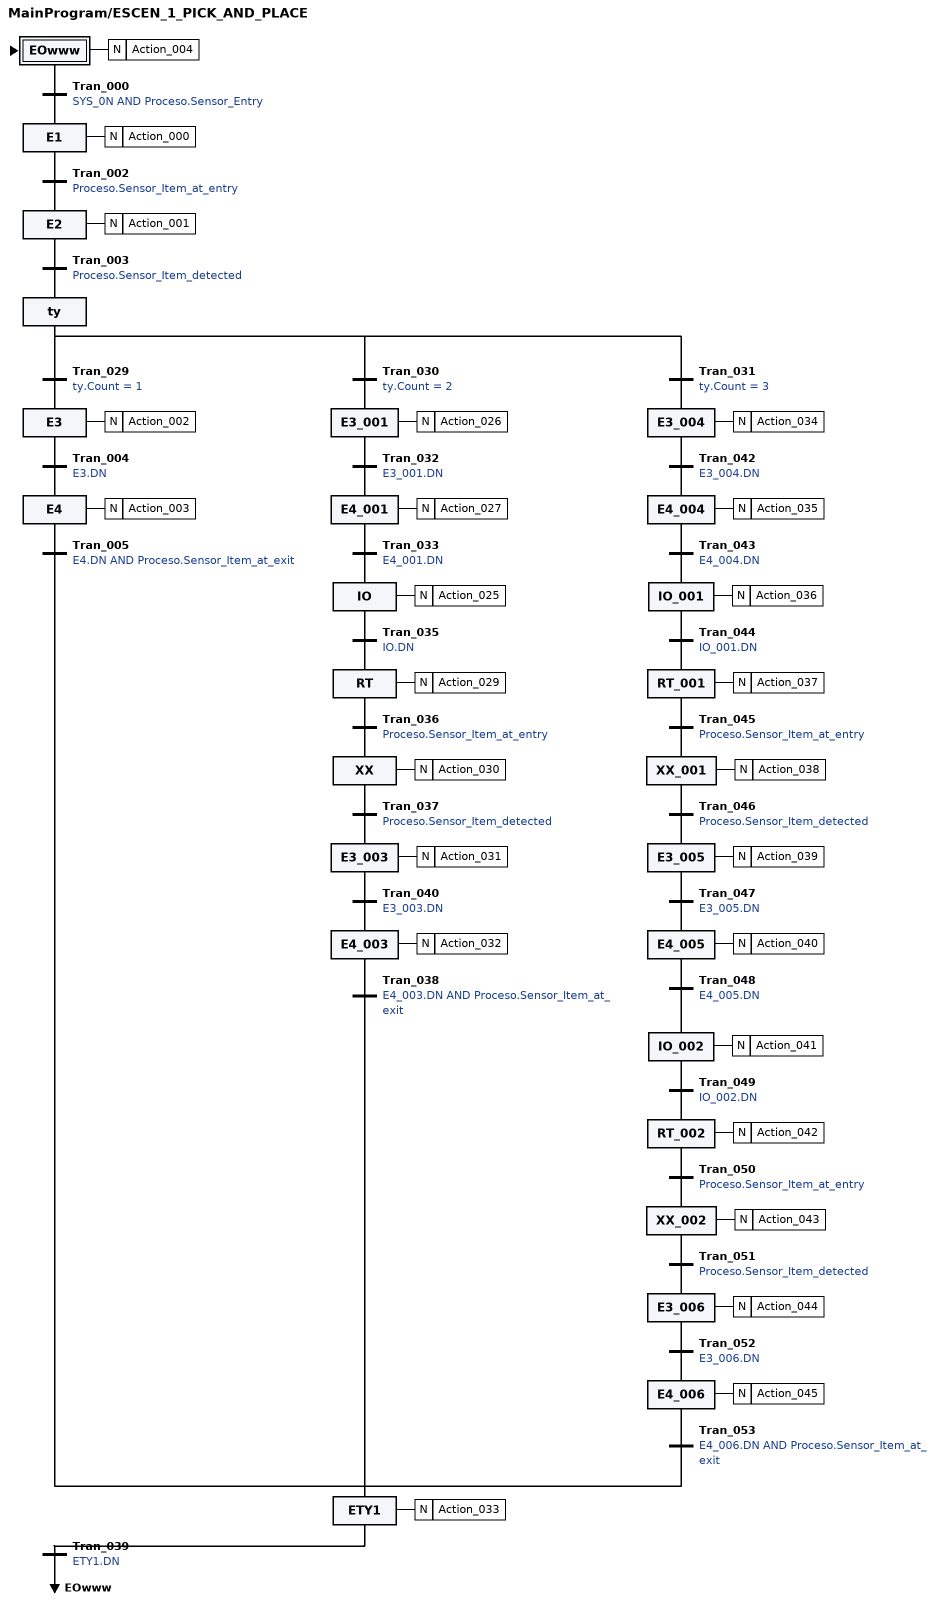
   INITIAL_STEP EOwww:
      ACTION Action_004 (N):
         Proceso.Cmd_Run_Grab:= 0;
         Proceso.Cmd_Run_Move_z:= 0;
         Proceso.Cmd_Run_Move_x:= 0;
         Proceso.Cmd_Run_Banda_Exit_conveyor:= 0;
         
      END_ACTION
   END_STEP
   TRANSITION Tran_000 FROM EOwww TO E1
      := SYS_0N AND Proceso.Sensor_Entry
   END_TRANSITION
   STEP E1:
      ACTION Action_000 (N):
         Proceso.Cmd_Run_Banda_Entry_Conveyor:= 1;
         
      END_ACTION
   END_STEP
   TRANSITION Tran_002 FROM E1 TO E2
      := Proceso.Sensor_Item_at_entry
   END_TRANSITION
   STEP E2:
      ACTION Action_001 (N):
         Proceso.Cmd_Run_Banda_Entry_Conveyor:= 0;
         Proceso.Cmd_Run_Move_z:= 1;
      END_ACTION
   END_STEP
   TRANSITION Tran_003 FROM E2 TO ty
      := Proceso.Sensor_Item_detected
   END_TRANSITION
   STEP ty:
   END_STEP
   TRANSITION Tran_029 FROM ty TO E3
      := ty.Count = 1
   END_TRANSITION
   TRANSITION Tran_030 FROM ty TO E3_001
      := ty.Count = 2
   END_TRANSITION
   TRANSITION Tran_031 FROM ty TO E3_004
      := ty.Count = 3
   END_TRANSITION
   STEP E3_001:
      ACTION Action_026 (N):
         
         Proceso.Cmd_Run_Grab:= 1;
         Proceso.Cmd_Run_Move_z:= 0;
         Proceso.Cmd_Run_Move_x:= 1;
         Proceso.Cmd_Run_Banda_Exit_conveyor:= 0;
      END_ACTION
   END_STEP
   STEP E3_004:
      ACTION Action_034 (N):
         
         Proceso.Cmd_Run_Grab:= 1;
         Proceso.Cmd_Run_Move_z:= 0;
         Proceso.Cmd_Run_Move_x:= 1;
         Proceso.Cmd_Run_Banda_Exit_conveyor:= 0;
      END_ACTION
   END_STEP
   STEP E3:
      ACTION Action_002 (N):
         
         Proceso.Cmd_Run_Grab:= 1;
         Proceso.Cmd_Run_Move_z:= 0;
         Proceso.Cmd_Run_Move_x:= 1;
         
      END_ACTION
   END_STEP
   TRANSITION Tran_004 FROM E3 TO E4
      := E3.DN
   END_TRANSITION
   TRANSITION Tran_032 FROM E3_001 TO E4_001
      := E3_001.DN
   END_TRANSITION
   TRANSITION Tran_042 FROM E3_004 TO E4_004
      := E3_004.DN
   END_TRANSITION
   STEP E4:
      ACTION Action_003 (N):
         Proceso.Cmd_Run_Move_z:= 1;
         
      END_ACTION
   END_STEP
   STEP E4_001:
      ACTION Action_027 (N):
         Proceso.Cmd_Run_Move_z:= 1;
         
      END_ACTION
   END_STEP
   STEP E4_004:
      ACTION Action_035 (N):
         Proceso.Cmd_Run_Move_z:= 1;
         
      END_ACTION
   END_STEP
   TRANSITION Tran_033 FROM E4_001 TO IO
      := E4_001.DN
   END_TRANSITION
   TRANSITION Tran_043 FROM E4_004 TO IO_001
      := E4_004.DN
   END_TRANSITION
   STEP IO:
      ACTION Action_025 (N):
         Proceso.Cmd_Run_Grab:= 0;
         Proceso.Cmd_Run_Move_z:= 0;
         Proceso.Cmd_Run_Move_x:= 0;
      END_ACTION
   END_STEP
   STEP IO_001:
      ACTION Action_036 (N):
         Proceso.Cmd_Run_Grab:= 0;
         Proceso.Cmd_Run_Move_z:= 0;
         Proceso.Cmd_Run_Move_x:= 0;
      END_ACTION
   END_STEP
   TRANSITION Tran_035 FROM IO TO RT
      := IO.DN
   END_TRANSITION
   STEP RT:
      ACTION Action_029 (N):
         Proceso.Cmd_Run_Banda_Entry_Conveyor:= 1;
      END_ACTION
   END_STEP
   TRANSITION Tran_044 FROM IO_001 TO RT_001
      := IO_001.DN
   END_TRANSITION
   TRANSITION Tran_036 FROM RT TO XX
      := Proceso.Sensor_Item_at_entry
   END_TRANSITION
   STEP RT_001:
      ACTION Action_037 (N):
         Proceso.Cmd_Run_Banda_Entry_Conveyor:= 1;
      END_ACTION
   END_STEP
   STEP XX:
      ACTION Action_030 (N):
         Proceso.Cmd_Run_Banda_Entry_Conveyor:= 0;
         Proceso.Cmd_Run_Move_z:= 1;
      END_ACTION
   END_STEP
   TRANSITION Tran_045 FROM RT_001 TO XX_001
      := Proceso.Sensor_Item_at_entry
   END_TRANSITION
   TRANSITION Tran_037 FROM XX TO E3_003
      := Proceso.Sensor_Item_detected
   END_TRANSITION
   STEP E3_003:
      ACTION Action_031 (N):
         
         Proceso.Cmd_Run_Grab:= 1;
         Proceso.Cmd_Run_Move_z:= 0;
         Proceso.Cmd_Run_Move_x:= 1;
         
      END_ACTION
   END_STEP
   STEP XX_001:
      ACTION Action_038 (N):
         Proceso.Cmd_Run_Banda_Entry_Conveyor:= 0;
         Proceso.Cmd_Run_Move_z:= 1;
      END_ACTION
   END_STEP
   TRANSITION Tran_040 FROM E3_003 TO E4_003
      := E3_003.DN
   END_TRANSITION
   TRANSITION Tran_046 FROM XX_001 TO E3_005
      := Proceso.Sensor_Item_detected
   END_TRANSITION
   STEP E3_005:
      ACTION Action_039 (N):
         
         Proceso.Cmd_Run_Grab:= 1;
         Proceso.Cmd_Run_Move_z:= 0;
         Proceso.Cmd_Run_Move_x:= 1;
         
      END_ACTION
   END_STEP
   STEP E4_003:
      ACTION Action_032 (N):
         Proceso.Cmd_Run_Move_z:= 1;
         
      END_ACTION
   END_STEP
   TRANSITION Tran_047 FROM E3_005 TO E4_005
      := E3_005.DN
   END_TRANSITION
   TRANSITION Tran_005 FROM E4 TO ETY1
      := E4.DN  AND Proceso.Sensor_Item_at_exit
   END_TRANSITION
   TRANSITION Tran_038 FROM E4_003 TO ETY1
      := E4_003.DN  AND Proceso.Sensor_Item_at_exit
   END_TRANSITION
   STEP E4_005:
      ACTION Action_040 (N):
         Proceso.Cmd_Run_Move_z:= 1;
         
      END_ACTION
   END_STEP
   TRANSITION Tran_048 FROM E4_005 TO IO_002
      := E4_005.DN
   END_TRANSITION
   STEP IO_002:
      ACTION Action_041 (N):
         Proceso.Cmd_Run_Grab:= 0;
         Proceso.Cmd_Run_Move_z:= 0;
         Proceso.Cmd_Run_Move_x:= 0;
      END_ACTION
   END_STEP
   TRANSITION Tran_049 FROM IO_002 TO RT_002
      := IO_002.DN
   END_TRANSITION
   STEP RT_002:
      ACTION Action_042 (N):
         Proceso.Cmd_Run_Banda_Entry_Conveyor:= 1;
      END_ACTION
   END_STEP
   TRANSITION Tran_050 FROM RT_002 TO XX_002
      := Proceso.Sensor_Item_at_entry
   END_TRANSITION
   STEP XX_002:
      ACTION Action_043 (N):
         Proceso.Cmd_Run_Banda_Entry_Conveyor:= 0;
         Proceso.Cmd_Run_Move_z:= 1;
      END_ACTION
   END_STEP
   TRANSITION Tran_051 FROM XX_002 TO E3_006
      := Proceso.Sensor_Item_detected
   END_TRANSITION
   STEP E3_006:
      ACTION Action_044 (N):
         
         Proceso.Cmd_Run_Grab:= 1;
         Proceso.Cmd_Run_Move_z:= 0;
         Proceso.Cmd_Run_Move_x:= 1;
         
      END_ACTION
   END_STEP
   TRANSITION Tran_052 FROM E3_006 TO E4_006
      := E3_006.DN
   END_TRANSITION
   STEP E4_006:
      ACTION Action_045 (N):
         Proceso.Cmd_Run_Move_z:= 1;
         ty.COUNT:=0;
         
      END_ACTION
   END_STEP
   TRANSITION Tran_053 FROM E4_006 TO ETY1
      := E4_006.DN AND Proceso.Sensor_Item_at_exit
   END_TRANSITION
   STEP ETY1:
      ACTION Action_033 (N):
         Proceso.Cmd_Run_Banda_Exit_conveyor:= 1;
         Proceso.Cmd_Run_Move_z:= 0;
         Proceso.Cmd_Run_Grab:= 0;
         Proceso.Cmd_Run_Move_x:= 0;
         
      END_ACTION
   END_STEP
   TRANSITION Tran_039 FROM ETY1 TO EOwww
      := ETY1.DN
   END_TRANSITION
END_ROUTINE

ROUTINE ESCEN_1_PICK_AND_PLACE_2   (* sequential function chart *)
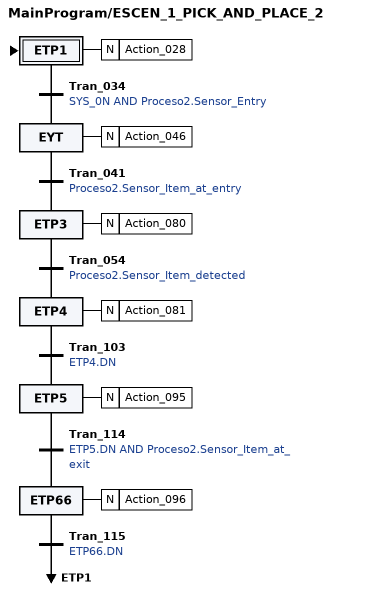
   INITIAL_STEP ETP1:
      ACTION Action_028 (N):
         Proceso2.Cmd_Run_Grab:= 0;
         Proceso2.Cmd_Run_Move_z:= 0;
         Proceso2.Cmd_Run_Move_x:= 0;
         Proceso2.Cmd_Run_Banda_Exit_conveyor:= 0;
         
      END_ACTION
   END_STEP
   TRANSITION Tran_034 FROM ETP1 TO EYT
      := SYS_0N AND Proceso2.Sensor_Entry
   END_TRANSITION
   STEP EYT:
      ACTION Action_046 (N):
         Proceso2.Cmd_Run_Banda_Entry_Conveyor:=1;
      END_ACTION
   END_STEP
   TRANSITION Tran_041 FROM EYT TO ETP3
      := Proceso2.Sensor_Item_at_entry
   END_TRANSITION
   STEP ETP3:
      ACTION Action_080 (N):
         Proceso2.Cmd_Run_Banda_Entry_Conveyor:= 0;
         Proceso2.Cmd_Run_Move_z:= 1;
      END_ACTION
   END_STEP
   TRANSITION Tran_054 FROM ETP3 TO ETP4
      := Proceso2.Sensor_Item_detected
   END_TRANSITION
   STEP ETP4:
      ACTION Action_081 (N):
         
         Proceso2.Cmd_Run_Grab:= 1;
         Proceso2.Cmd_Run_Move_z:= 0;
         Proceso2.Cmd_Run_Move_x:= 1;
         
      END_ACTION
   END_STEP
   TRANSITION Tran_103 FROM ETP4 TO ETP5
      := ETP4.DN
   END_TRANSITION
   STEP ETP5:
      ACTION Action_095 (N):
         Proceso2.Cmd_Run_Move_z:= 1;
         
      END_ACTION
   END_STEP
   TRANSITION Tran_114 FROM ETP5 TO ETP66
      := ETP5.DN  AND Proceso2.Sensor_Item_at_exit
   END_TRANSITION
   STEP ETP66:
      ACTION Action_096 (N):
         Proceso2.Cmd_Run_Banda_Exit_conveyor:= 1;
         Proceso2.Cmd_Run_Move_z:= 0;
         Proceso2.Cmd_Run_Grab:= 0;
         Proceso2.Cmd_Run_Move_x:= 0;
         
      END_ACTION
   END_STEP
   TRANSITION Tran_115 FROM ETP66 TO ETP1
      := ETP66.DN
   END_TRANSITION
END_ROUTINE

ROUTINE ESCENA_3_LINE_1   (* sequential function chart *)
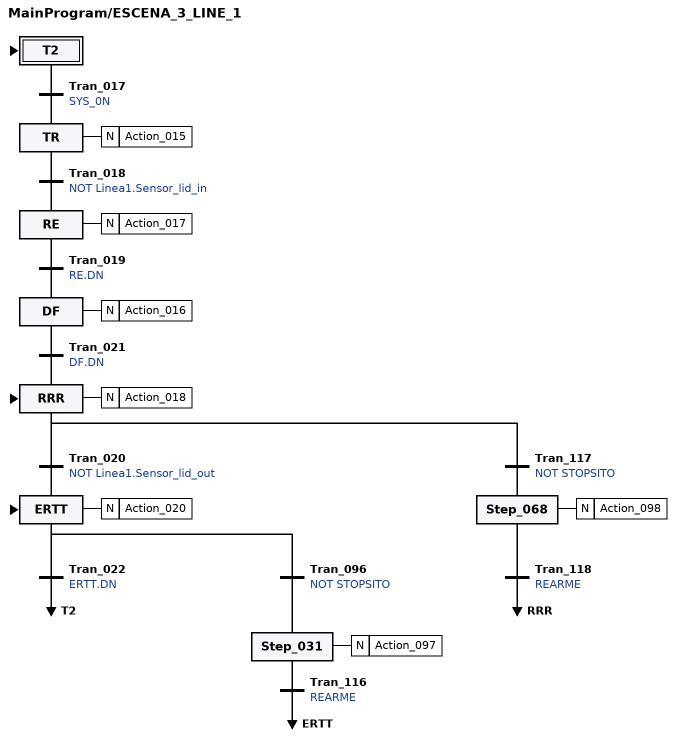
   INITIAL_STEP T2:
   END_STEP
   TRANSITION Tran_017 FROM T2 TO TR
      := SYS_0N
   END_TRANSITION
   STEP TR:
      ACTION Action_015 (N):
         Linea1.Cmd_Run_Banda_Lids_In:=1;
      END_ACTION
   END_STEP
   TRANSITION Tran_018 FROM TR TO RE
      := NOT Linea1.Sensor_lid_in
   END_TRANSITION
   STEP RE:
      ACTION Action_017 (N):
         Linea1.Cmd_Run_Banda_Lids_In:=1;
      END_ACTION
   END_STEP
   TRANSITION Tran_019 FROM RE TO DF
      := RE.DN
   END_TRANSITION
   STEP DF:
      ACTION Action_016 (N):
         Linea1.Cmd_Run_Banda_Lids_In:=0;
      END_ACTION
   END_STEP
   TRANSITION Tran_021 FROM DF TO RRR
      := DF.DN
   END_TRANSITION
   STEP RRR:
      ACTION Action_018 (N):
         Linea1.Cmd_Run_Brazo:=1;
         Linea1.Cmd_Run_Banda_Lids_In:=0;
      END_ACTION
   END_STEP
   TRANSITION Tran_117 FROM RRR TO Step_068
      := NOT STOPSITO
   END_TRANSITION
   STEP Step_068:
      ACTION Action_098 (N):
         Linea1.Cmd_Run_Banda_Lids_Out1:=0;
         Linea1.Cmd_Run_Banda_Lids_Out2:=0;
         Linea1.Cmd_Run_Brazo:=0;
         Linea1.Cmd_Run_Banda_Lids_In:=0;
      END_ACTION
   END_STEP
   TRANSITION Tran_118 FROM Step_068 TO RRR
      := REARME
   END_TRANSITION
   TRANSITION Tran_020 FROM RRR TO ERTT
      := NOT Linea1.Sensor_lid_out
   END_TRANSITION
   STEP ERTT:
      ACTION Action_020 (N):
         Linea1.Cmd_Run_Banda_Lids_Out1:=1;
         Linea1.Cmd_Run_Banda_Lids_Out2:=1;
      END_ACTION
   END_STEP
   TRANSITION Tran_096 FROM ERTT TO Step_031
      := NOT STOPSITO
   END_TRANSITION
   STEP Step_031:
      ACTION Action_097 (N):
         Linea1.Cmd_Run_Banda_Lids_Out1:=0;
         Linea1.Cmd_Run_Banda_Lids_Out2:=0;
         Linea1.Cmd_Run_Brazo:=0;
         Linea1.Cmd_Run_Banda_Lids_In:=0;
      END_ACTION
   END_STEP
   TRANSITION Tran_022 FROM ERTT TO T2
      := ERTT.DN
   END_TRANSITION
   TRANSITION Tran_116 FROM Step_031 TO ERTT
      := REARME
   END_TRANSITION
END_ROUTINE

ROUTINE ESCENA_3_LINE_2   (* sequential function chart *)
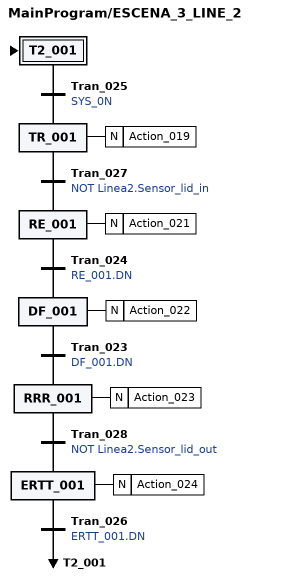
   INITIAL_STEP T2_001:
   END_STEP
   TRANSITION Tran_025 FROM T2_001 TO TR_001
      := SYS_0N
   END_TRANSITION
   STEP TR_001:
      ACTION Action_019 (N):
         Linea2.Cmd_Run_Banda_Lids_In:=1;
      END_ACTION
   END_STEP
   TRANSITION Tran_027 FROM TR_001 TO RE_001
      := NOT Linea2.Sensor_lid_in
   END_TRANSITION
   STEP RE_001:
      ACTION Action_021 (N):
         Linea2.Cmd_Run_Banda_Lids_In:=1;
      END_ACTION
   END_STEP
   TRANSITION Tran_024 FROM RE_001 TO DF_001
      := RE_001.DN
   END_TRANSITION
   STEP DF_001:
      ACTION Action_022 (N):
         Linea2.Cmd_Run_Banda_Lids_In:=0;
      END_ACTION
   END_STEP
   TRANSITION Tran_023 FROM DF_001 TO RRR_001
      := DF_001.DN
   END_TRANSITION
   STEP RRR_001:
      ACTION Action_023 (N):
         Linea2.Cmd_Run_Brazo:=1;
         Linea2.Cmd_Run_Banda_Lids_In:=0;
      END_ACTION
   END_STEP
   TRANSITION Tran_028 FROM RRR_001 TO ERTT_001
      := NOT Linea2.Sensor_lid_out
   END_TRANSITION
   STEP ERTT_001:
      ACTION Action_024 (N):
         Linea2.Cmd_Run_Banda_Lids_Out1:=1;
         Linea2.Cmd_Run_Banda_Lids_Out2:=1;
      END_ACTION
   END_STEP
   TRANSITION Tran_026 FROM ERTT_001 TO T2_001
      := ERTT_001.DN
   END_TRANSITION
END_ROUTINE

ROUTINE ESCENA_3_LINE_3   (* sequential function chart *)
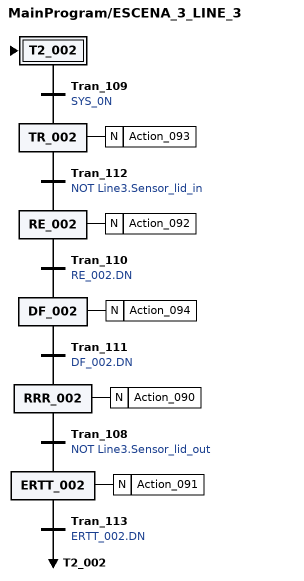
   INITIAL_STEP T2_002:
   END_STEP
   TRANSITION Tran_109 FROM T2_002 TO TR_002
      := SYS_0N
   END_TRANSITION
   STEP TR_002:
      ACTION Action_093 (N):
         Line3.Cmd_Run_Banda_Lids_In:=1;
      END_ACTION
   END_STEP
   TRANSITION Tran_112 FROM TR_002 TO RE_002
      := NOT Line3.Sensor_lid_in
   END_TRANSITION
   STEP RE_002:
      ACTION Action_092 (N):
         Line3.Cmd_Run_Banda_Lids_In:=1;
      END_ACTION
   END_STEP
   TRANSITION Tran_110 FROM RE_002 TO DF_002
      := RE_002.DN
   END_TRANSITION
   STEP DF_002:
      ACTION Action_094 (N):
         Line3.Cmd_Run_Banda_Lids_In:=0;
      END_ACTION
   END_STEP
   TRANSITION Tran_111 FROM DF_002 TO RRR_002
      := DF_002.DN
   END_TRANSITION
   STEP RRR_002:
      ACTION Action_090 (N):
         Line3.Cmd_Run_Brazo:=1;
         Line3.Cmd_Run_Banda_Lids_In:=0;
      END_ACTION
   END_STEP
   TRANSITION Tran_108 FROM RRR_002 TO ERTT_002
      := NOT Line3.Sensor_lid_out
   END_TRANSITION
   STEP ERTT_002:
      ACTION Action_091 (N):
         Line3.Cmd_Run_Banda_Lids_Out1:=1;
         Line3.Cmd_Run_Banda_Lids_Out2:=1;
      END_ACTION
   END_STEP
   TRANSITION Tran_113 FROM ERTT_002 TO T2_002
      := ERTT_002.DN
   END_TRANSITION
END_ROUTINE

ROUTINE ESCENA_4_XYZ   (* sequential function chart *)
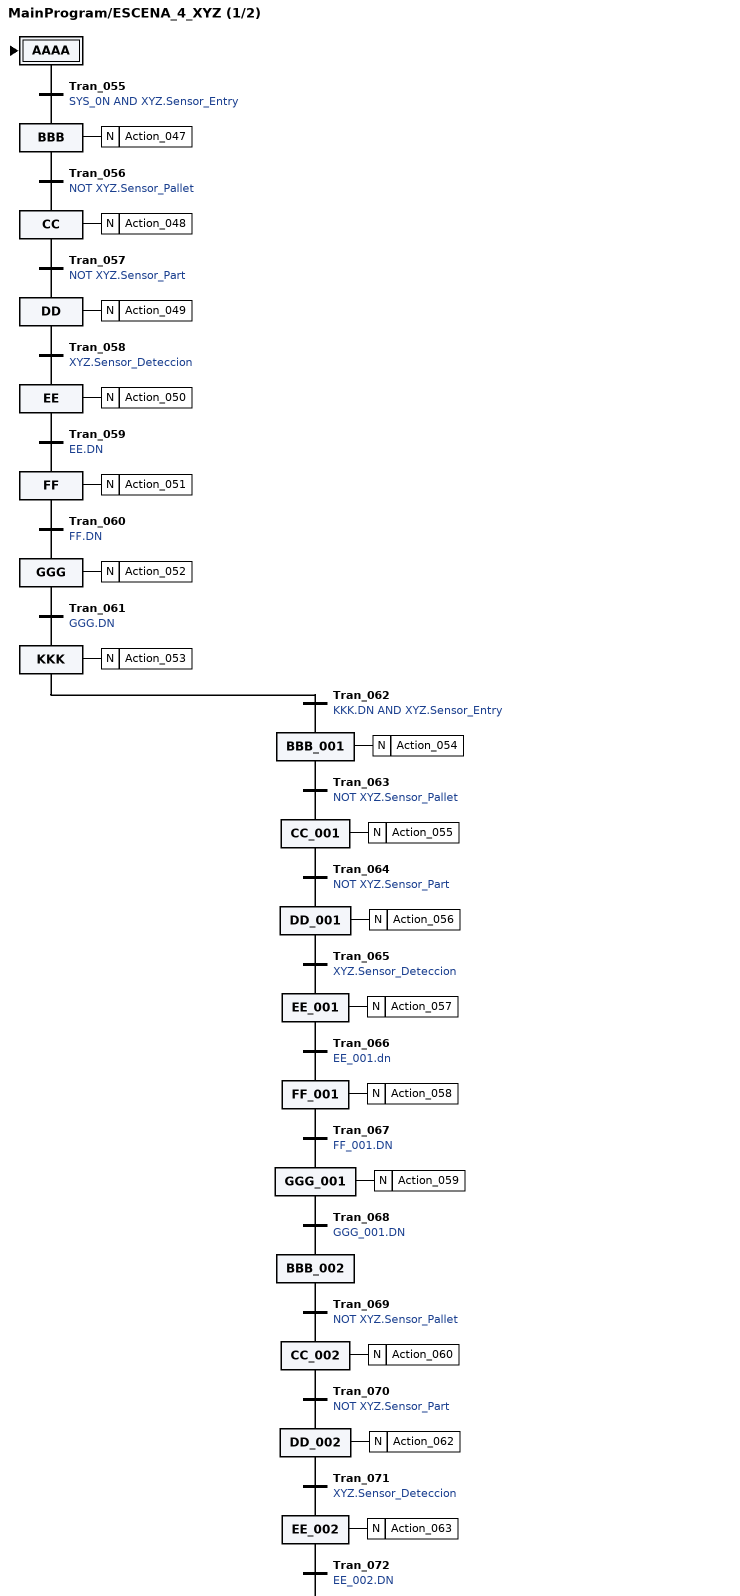
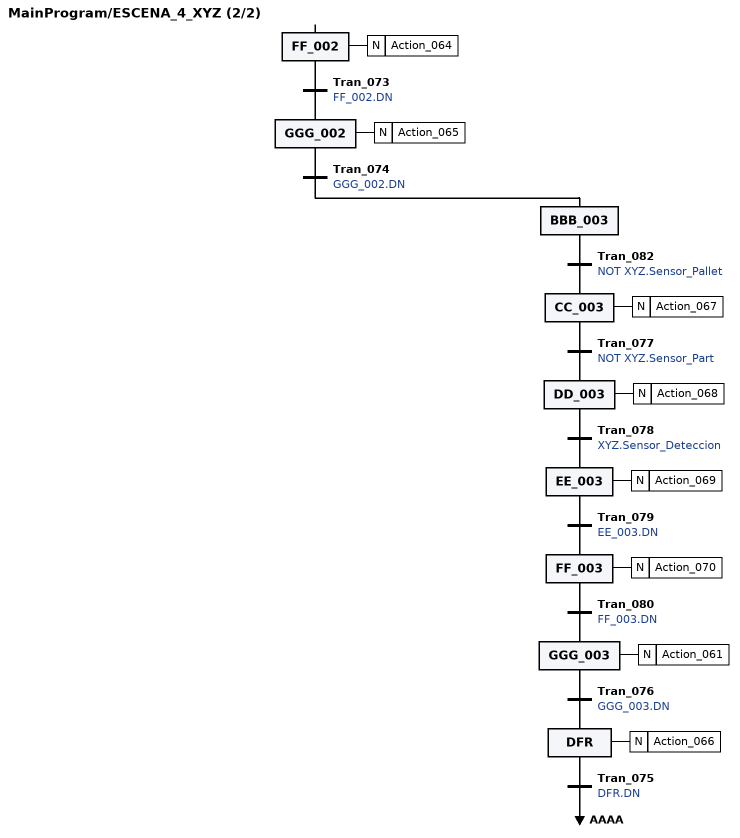
   INITIAL_STEP AAAA:
   END_STEP
   TRANSITION Tran_055 FROM AAAA TO BBB
      := SYS_0N AND XYZ.Sensor_Entry
   END_TRANSITION
   STEP BBB:
      ACTION Action_047 (N):
         XYZ.Cmd_Run_Pallet_conveyor:=1;
         XYZ.Cmd_Run_Part_conveyor:=1;
         XYZ.Cmd_Run_Emiter_Pallets:=1;
         
      END_ACTION
   END_STEP
   TRANSITION Tran_056 FROM BBB TO CC
      := NOT XYZ.Sensor_Pallet
   END_TRANSITION
   STEP CC:
      ACTION Action_048 (N):
         XYZ.Cmd_Run_Pallet_conveyor:=0;
         XYZ.Cmd_Run_Emiter_Pallets:=0;
         
      END_ACTION
   END_STEP
   TRANSITION Tran_057 FROM CC TO DD
      := NOT XYZ.Sensor_Part
   END_TRANSITION
   STEP DD:
      ACTION Action_049 (N):
         XYZ.Cmd_Run_Part_conveyor:=0;
         
         XYZ.V_eje_X:=7.7;
         XYZ.V_eje_Y:=5.4;
         XYZ.V_eje_Z:=8.5;
         
         
      END_ACTION
   END_STEP
   TRANSITION Tran_058 FROM DD TO EE
      := XYZ.Sensor_Deteccion
   END_TRANSITION
   STEP EE:
      ACTION Action_050 (N):
         XYZ.Cmd_Run_GradXYZ:=1;
         XYZ.V_eje_Z:=3;
         
      END_ACTION
   END_STEP
   TRANSITION Tran_059 FROM EE TO FF
      := EE.DN
   END_TRANSITION
   STEP FF:
      ACTION Action_051 (N):
         
         XYZ.Cmd_Run_GradXYZ:=1;
         XYZ.V_eje_X:=3.1;
         XYZ.V_eje_Z:=10;
         
         
         
      END_ACTION
   END_STEP
   TRANSITION Tran_060 FROM FF TO GGG
      := FF.DN
   END_TRANSITION
   STEP GGG:
      ACTION Action_052 (N):
         XYZ.Cmd_Run_GradXYZ:=0;
         
         
      END_ACTION
   END_STEP
   TRANSITION Tran_061 FROM GGG TO KKK
      := GGG.DN
   END_TRANSITION
   STEP KKK:
      ACTION Action_053 (N):
         XYZ.Cmd_Run_Pallet_conveyor:=1;
         
      END_ACTION
   END_STEP
   TRANSITION Tran_062 FROM KKK TO BBB_001
      := KKK.DN AND XYZ.Sensor_Entry
   END_TRANSITION
   STEP BBB_001:
      ACTION Action_054 (N):
         XYZ.Cmd_Run_Pallet_conveyor:=1;
         XYZ.Cmd_Run_Part_conveyor:=1;
         XYZ.Cmd_Run_Emiter_Pallets:=1;
      END_ACTION
   END_STEP
   TRANSITION Tran_063 FROM BBB_001 TO CC_001
      := NOT XYZ.Sensor_Pallet
   END_TRANSITION
   STEP CC_001:
      ACTION Action_055 (N):
         XYZ.Cmd_Run_Pallet_conveyor:=0;
         XYZ.Cmd_Run_Emiter_Pallets:=0;
         
      END_ACTION
   END_STEP
   TRANSITION Tran_064 FROM CC_001 TO DD_001
      := NOT XYZ.Sensor_Part
   END_TRANSITION
   STEP DD_001:
      ACTION Action_056 (N):
         XYZ.Cmd_Run_Part_conveyor:=0;
         XYZ.Cmd_Run_Emiter_Pallets:=0;
         XYZ.V_eje_X:=7.7;
         XYZ.V_eje_Y:=5.4;
         XYZ.V_eje_Z:=8.5;
      END_ACTION
   END_STEP
   TRANSITION Tran_065 FROM DD_001 TO EE_001
      := XYZ.Sensor_Deteccion
   END_TRANSITION
   STEP EE_001:
      ACTION Action_057 (N):
         XYZ.Cmd_Run_GradXYZ:=1;
         XYZ.V_eje_Z:=3;
      END_ACTION
   END_STEP
   TRANSITION Tran_066 FROM EE_001 TO FF_001
      := EE_001.dn
   END_TRANSITION
   STEP FF_001:
      ACTION Action_058 (N):
         XYZ.Cmd_Run_GradXYZ:=1;
         XYZ.V_eje_X:=3.1;
         XYZ.V_eje_Z:=10;
      END_ACTION
   END_STEP
   TRANSITION Tran_067 FROM FF_001 TO GGG_001
      := FF_001.DN
   END_TRANSITION
   STEP GGG_001:
      ACTION Action_059 (N):
         XYZ.Cmd_Run_GradXYZ:=0;
      END_ACTION
   END_STEP
   TRANSITION Tran_068 FROM GGG_001 TO BBB_002
      := GGG_001.DN
   END_TRANSITION
   STEP BBB_002:
   END_STEP
   TRANSITION Tran_069 FROM BBB_002 TO CC_002
      := NOT XYZ.Sensor_Pallet
   END_TRANSITION
   STEP CC_002:
      ACTION Action_060 (N):
         XYZ.Cmd_Run_Pallet_conveyor:=0;
         XYZ.Cmd_Run_Part_conveyor:=1;
      END_ACTION
   END_STEP
   TRANSITION Tran_070 FROM CC_002 TO DD_002
      := NOT XYZ.Sensor_Part
   END_TRANSITION
   STEP DD_002:
      ACTION Action_062 (N):
         XYZ.Cmd_Run_Part_conveyor:=0;
         XYZ.V_eje_X:=7.7;
         XYZ.V_eje_Y:=5.4;
         XYZ.V_eje_Z:=8.5;
         
      END_ACTION
   END_STEP
   TRANSITION Tran_071 FROM DD_002 TO EE_002
      := XYZ.Sensor_Deteccion
   END_TRANSITION
   STEP EE_002:
      ACTION Action_063 (N):
         XYZ.Cmd_Run_GradXYZ:=1;
         XYZ.V_eje_Z:=3;
      END_ACTION
   END_STEP
   TRANSITION Tran_072 FROM EE_002 TO FF_002
      := EE_002.DN
   END_TRANSITION
   STEP FF_002:
      ACTION Action_064 (N):
         XYZ.Cmd_Run_GradXYZ:=1;
         XYZ.V_eje_X:=3.1;
         XYZ.V_eje_Z:=10;
      END_ACTION
   END_STEP
   TRANSITION Tran_073 FROM FF_002 TO GGG_002
      := FF_002.DN
   END_TRANSITION
   STEP GGG_002:
      ACTION Action_065 (N):
         XYZ.Cmd_Run_GradXYZ:=0;
         
      END_ACTION
   END_STEP
   TRANSITION Tran_074 FROM GGG_002 TO BBB_003
      := GGG_002.DN
   END_TRANSITION
   STEP BBB_003:
   END_STEP
   TRANSITION Tran_082 FROM BBB_003 TO CC_003
      := NOT XYZ.Sensor_Pallet
   END_TRANSITION
   STEP CC_003:
      ACTION Action_067 (N):
         XYZ.Cmd_Run_Pallet_conveyor:=0;
         XYZ.Cmd_Run_Part_conveyor:=1;
      END_ACTION
   END_STEP
   TRANSITION Tran_077 FROM CC_003 TO DD_003
      := NOT XYZ.Sensor_Part
   END_TRANSITION
   STEP DD_003:
      ACTION Action_068 (N):
         XYZ.Cmd_Run_Part_conveyor:=0;
         XYZ.V_eje_X:=7.7;
         XYZ.V_eje_Y:=5.4;
         XYZ.V_eje_Z:=8.5;
         
      END_ACTION
   END_STEP
   TRANSITION Tran_078 FROM DD_003 TO EE_003
      := XYZ.Sensor_Deteccion
   END_TRANSITION
   STEP EE_003:
      ACTION Action_069 (N):
         XYZ.Cmd_Run_GradXYZ:=1;
         XYZ.V_eje_Z:=3;
      END_ACTION
   END_STEP
   TRANSITION Tran_079 FROM EE_003 TO FF_003
      := EE_003.DN
   END_TRANSITION
   STEP FF_003:
      ACTION Action_070 (N):
         XYZ.Cmd_Run_GradXYZ:=1;
         XYZ.V_eje_X:=3.1;
         XYZ.V_eje_Z:=10;
      END_ACTION
   END_STEP
   TRANSITION Tran_080 FROM FF_003 TO GGG_003
      := FF_003.DN
   END_TRANSITION
   STEP GGG_003:
      ACTION Action_061 (N):
         XYZ.Cmd_Run_GradXYZ:=0;
         
         
      END_ACTION
   END_STEP
   TRANSITION Tran_076 FROM GGG_003 TO DFR
      := GGG_003.DN
   END_TRANSITION
   STEP DFR:
      ACTION Action_066 (N):
         XYZ.Cmd_Run_Pallet_conveyor:=1;
      END_ACTION
   END_STEP
   TRANSITION Tran_075 FROM DFR TO AAAA
      := DFR.DN
   END_TRANSITION
END_ROUTINE

ROUTINE ESCENA_5_HIGH   (* sequential function chart *)
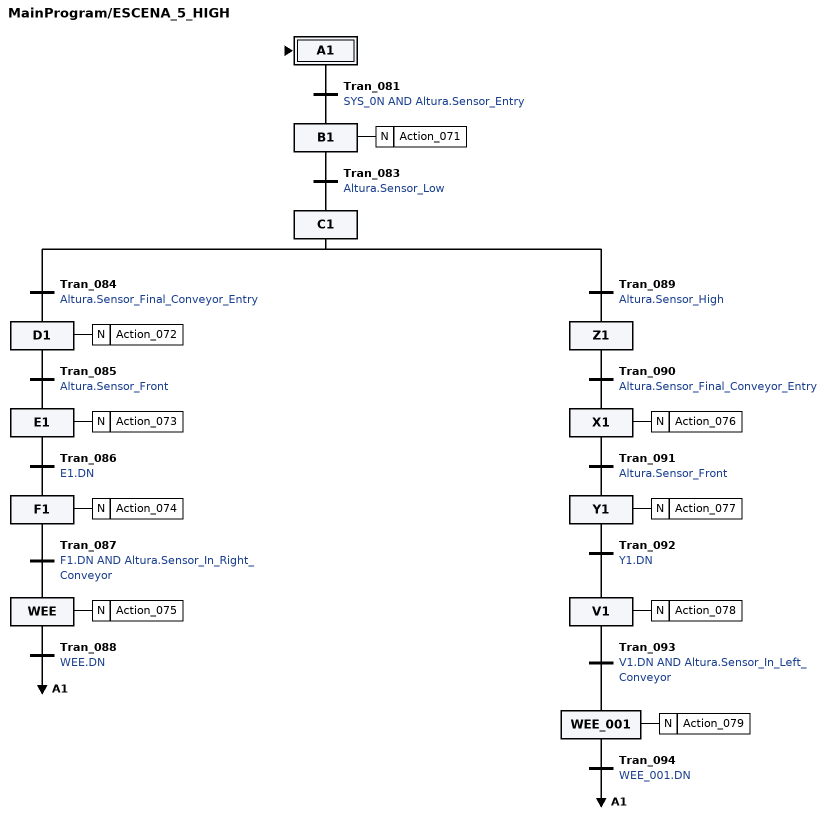
   INITIAL_STEP A1:
   END_STEP
   TRANSITION Tran_081 FROM A1 TO B1
      := SYS_0N AND Altura.Sensor_Entry
   END_TRANSITION
   STEP B1:
      ACTION Action_071 (N):
         Altura.Cmd_Run_Conveyor_Entry:=1;
      END_ACTION
   END_STEP
   TRANSITION Tran_083 FROM B1 TO C1
      := Altura.Sensor_Low
   END_TRANSITION
   STEP C1:
   END_STEP
   TRANSITION Tran_084 FROM C1 TO D1
      := Altura.Sensor_Final_Conveyor_Entry
   END_TRANSITION
   TRANSITION Tran_089 FROM C1 TO Z1
      := Altura.Sensor_High
   END_TRANSITION
   STEP D1:
      ACTION Action_072 (N):
         Altura.Cmd_Run_Conveyor_Entry:=1;
         Altura.Cmd_Run_Load:=1;
      END_ACTION
   END_STEP
   STEP Z1:
   END_STEP
   TRANSITION Tran_085 FROM D1 TO E1
      := Altura.Sensor_Front
   END_TRANSITION
   TRANSITION Tran_090 FROM Z1 TO X1
      := Altura.Sensor_Final_Conveyor_Entry
   END_TRANSITION
   STEP E1:
      ACTION Action_073 (N):
         Altura.Cmd_Run_Load:=0;
         Altura.Cmd_Run_Turn:=1;
         Altura.Cmd_Run_Conveyor_Entry:=0;
         
      END_ACTION
   END_STEP
   STEP X1:
      ACTION Action_076 (N):
         Altura.Cmd_Run_Conveyor_Entry:=1;
         Altura.Cmd_Run_Load:=1;
      END_ACTION
   END_STEP
   TRANSITION Tran_086 FROM E1 TO F1
      := E1.DN
   END_TRANSITION
   TRANSITION Tran_091 FROM X1 TO Y1
      := Altura.Sensor_Front
   END_TRANSITION
   STEP F1:
      ACTION Action_074 (N):
         Altura.Cmd_Run_Un_Load:=1;
         Altura.Cmd_Run_Conveyor_Right:=1;
         
         
      END_ACTION
   END_STEP
   TRANSITION Tran_087 FROM F1 TO WEE
      := F1.DN AND Altura.Sensor_In_Right_Conveyor
   END_TRANSITION
   STEP Y1:
      ACTION Action_077 (N):
         Altura.Cmd_Run_Load:=0;
         Altura.Cmd_Run_Turn:=1;
         Altura.Cmd_Run_Conveyor_Entry:=0;
         
      END_ACTION
   END_STEP
   STEP WEE:
      ACTION Action_075 (N):
         Altura.Cmd_Run_Un_Load:=0;
         Altura.Cmd_Run_Conveyor_Right:=1;
         Altura.Cmd_Run_Turn:=0;
         
      END_ACTION
   END_STEP
   TRANSITION Tran_092 FROM Y1 TO V1
      := Y1.DN
   END_TRANSITION
   TRANSITION Tran_088 FROM WEE TO A1
      := WEE.DN
   END_TRANSITION
   STEP V1:
      ACTION Action_078 (N):
         Altura.Cmd_Run_Load:=1;
         Altura.Cmd_Run_Conveyor_Left:=1;
         
      END_ACTION
   END_STEP
   TRANSITION Tran_093 FROM V1 TO WEE_001
      := V1.DN AND Altura.Sensor_In_Left_Conveyor
   END_TRANSITION
   STEP WEE_001:
      ACTION Action_079 (N):
         Altura.Cmd_Run_Load:=0;
         Altura.Cmd_Run_Conveyor_Left:=1;
         Altura.Cmd_Run_Turn:=0;
         
      END_ACTION
   END_STEP
   TRANSITION Tran_094 FROM WEE_001 TO A1
      := WEE_001.DN
   END_TRANSITION
END_ROUTINE

ROUTINE ESCENA_6_WEIGHT   (* sequential function chart *)
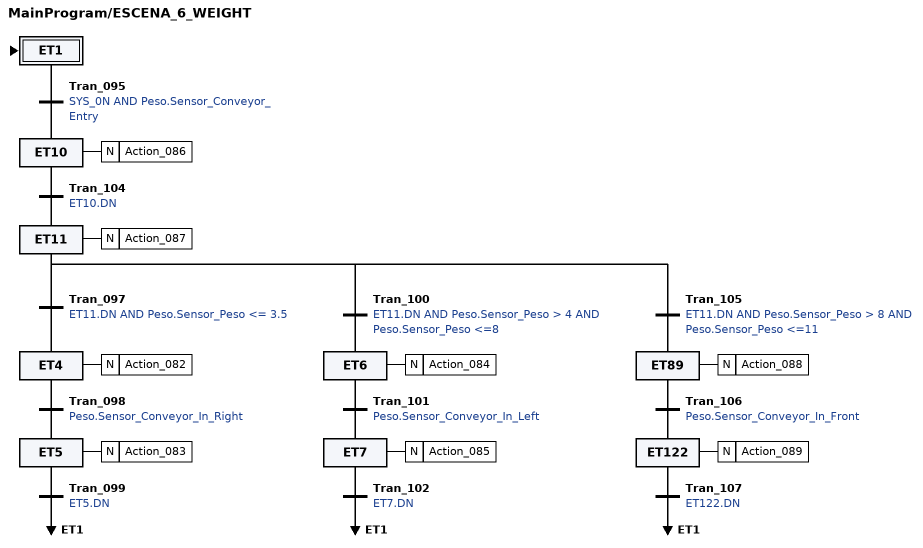
   INITIAL_STEP ET1:
   END_STEP
   TRANSITION Tran_095 FROM ET1 TO ET10
      := SYS_0N AND Peso.Sensor_Conveyor_Entry
   END_TRANSITION
   STEP ET10:
      ACTION Action_086 (N):
         Peso.Cmd_Run_Conveyor_Peso:=1;
         
      END_ACTION
   END_STEP
   TRANSITION Tran_104 FROM ET10 TO ET11
      := ET10.DN
   END_TRANSITION
   STEP ET11:
      ACTION Action_087 (N):
         Peso.Cmd_Run_Conveyor_Peso:=0;
         
      END_ACTION
   END_STEP
   TRANSITION Tran_097 FROM ET11 TO ET4
      := ET11.DN AND Peso.Sensor_Peso <= 3.5
   END_TRANSITION
   TRANSITION Tran_100 FROM ET11 TO ET6
      := ET11.DN AND  Peso.Sensor_Peso > 4  AND Peso.Sensor_Peso <=8
   END_TRANSITION
   TRANSITION Tran_105 FROM ET11 TO ET89
      := ET11.DN AND  Peso.Sensor_Peso > 8  AND Peso.Sensor_Peso <=11
   END_TRANSITION
   STEP ET89:
      ACTION Action_088 (N):
         Peso.Cmd_Run_Conveyor_Peso:=1;
         Peso.Cmd_Run_Send_Adelante:=1;
      END_ACTION
   END_STEP
   STEP ET6:
      ACTION Action_084 (N):
         Peso.Cmd_Run_Conveyor_Peso:=1;
         Peso.Cmd_Run_Send_Left:=1;
         Peso.Cmd_Run_Send_Adelante:=1;
      END_ACTION
   END_STEP
   STEP ET4:
      ACTION Action_082 (N):
         Peso.Cmd_Run_Conveyor_Peso:=1;
         Peso.Cmd_Run_Send_Right:=1;
         Peso.Cmd_Run_Send_Adelante:=1;
      END_ACTION
   END_STEP
   TRANSITION Tran_106 FROM ET89 TO ET122
      := Peso.Sensor_Conveyor_In_Front
   END_TRANSITION
   TRANSITION Tran_101 FROM ET6 TO ET7
      := Peso.Sensor_Conveyor_In_Left
   END_TRANSITION
   TRANSITION Tran_098 FROM ET4 TO ET5
      := Peso.Sensor_Conveyor_In_Right
   END_TRANSITION
   STEP ET122:
      ACTION Action_089 (N):
         Peso.Cmd_Run_Conveyor_Front:=1;
         Peso.Cmd_Run_Conveyor_Peso:=0;
         Peso.Cmd_Run_Send_Adelante:=0;
         
      END_ACTION
   END_STEP
   STEP ET7:
      ACTION Action_085 (N):
         Peso.Cmd_Run_Conveyor_Left:=1;
         Peso.Cmd_Run_Conveyor_Peso:=0;
         Peso.Cmd_Run_Send_Adelante:=0;
         Peso.Cmd_Run_Send_Left:=0;
         
      END_ACTION
   END_STEP
   STEP ET5:
      ACTION Action_083 (N):
         Peso.Cmd_Run_Conveyor_Right:=1;
         Peso.Cmd_Run_Conveyor_Peso:=0;
         Peso.Cmd_Run_Send_Adelante:=0;
         Peso.Cmd_Run_Send_Right:=0;
         
      END_ACTION
   END_STEP
   TRANSITION Tran_107 FROM ET122 TO ET1
      := ET122.DN
   END_TRANSITION
   TRANSITION Tran_099 FROM ET5 TO ET1
      := ET5.DN
   END_TRANSITION
   TRANSITION Tran_102 FROM ET7 TO ET1
      := ET7.DN
   END_TRANSITION
END_ROUTINE

ROUTINE ESCENE_2_SEPARATIO   (* sequential function chart *)
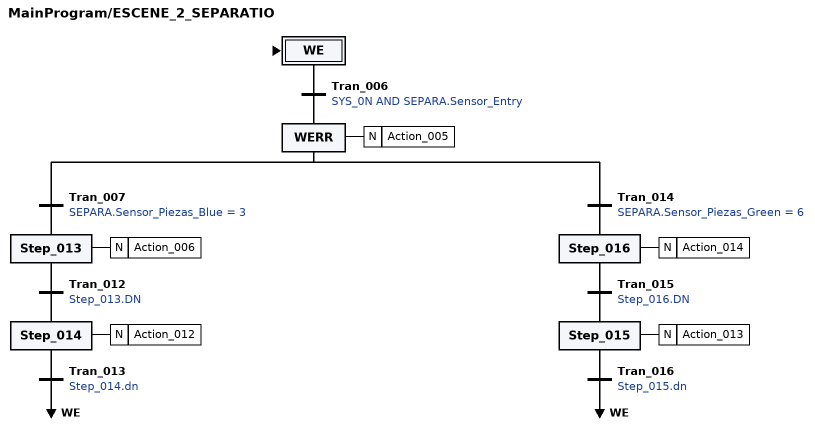
   INITIAL_STEP WE:
   END_STEP
   TRANSITION Tran_006 FROM WE TO WERR
      := SYS_0N AND SEPARA.Sensor_Entry
   END_TRANSITION
   STEP WERR:
      ACTION Action_005 (N):
         
         SEPARA.Cmd_Run_Banda_Conveyor:=1;
      END_ACTION
   END_STEP
   TRANSITION Tran_007 FROM WERR TO Step_013
      := 
         SEPARA.Sensor_Piezas_Blue = 3
   END_TRANSITION
   TRANSITION Tran_014 FROM WERR TO Step_016
      := SEPARA.Sensor_Piezas_Green = 6
   END_TRANSITION
   STEP Step_013:
      ACTION Action_006 (N):
         SEPARA.Cmd_Run_Pusher_Blue:=1;
         SEPARA.Cmd_Run_Banda_Conveyor:=0;
      END_ACTION
   END_STEP
   STEP Step_016:
      ACTION Action_014 (N):
         SEPARA.Cmd_Run_Pusher_Green:=1;
         SEPARA.Cmd_Run_Banda_Conveyor:=0;
      END_ACTION
   END_STEP
   TRANSITION Tran_012 FROM Step_013 TO Step_014
      := Step_013.DN
   END_TRANSITION
   TRANSITION Tran_015 FROM Step_016 TO Step_015
      := Step_016.DN
   END_TRANSITION
   STEP Step_014:
      ACTION Action_012 (N):
         SEPARA.Cmd_Run_Pusher_Blue:=0;
         
      END_ACTION
   END_STEP
   STEP Step_015:
      ACTION Action_013 (N):
         SEPARA.Cmd_Run_Pusher_Green:=0;
      END_ACTION
   END_STEP
   TRANSITION Tran_013 FROM Step_014 TO WE
      := Step_014.dn
   END_TRANSITION
   TRANSITION Tran_016 FROM Step_015 TO WE
      := Step_015.dn
   END_TRANSITION
END_ROUTINE

ROUTINE MainRoutine   (* ladder *)
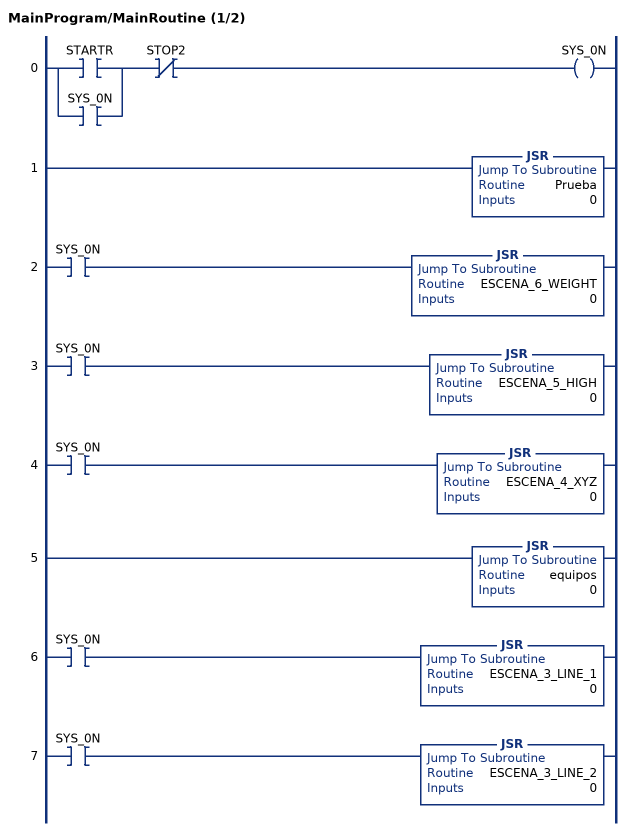
   0: [XIC(STARTR) ,XIC(SYS_0N) ]XIO(STOP2)OTE(SYS_0N);
   1: JSR(Prueba,0);
   2: XIC(SYS_0N)JSR(ESCENA_6_WEIGHT,0);
   3: XIC(SYS_0N)JSR(ESCENA_5_HIGH,0);
   4: XIC(SYS_0N)JSR(ESCENA_4_XYZ,0);
   5: JSR(equipos,0);
   6: XIC(SYS_0N)JSR(ESCENA_3_LINE_1,0);
   7: XIC(SYS_0N)JSR(ESCENA_3_LINE_2,0);
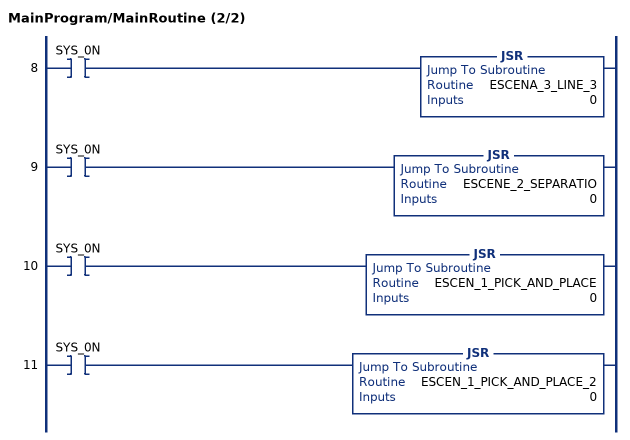
   8: XIC(SYS_0N)JSR(ESCENA_3_LINE_3,0);
   9: XIC(SYS_0N)JSR(ESCENE_2_SEPARATIO,0);
   10: XIC(SYS_0N)JSR(ESCEN_1_PICK_AND_PLACE,0);
   11: XIC(SYS_0N)JSR(ESCEN_1_PICK_AND_PLACE_2,0);
END_ROUTINE

ROUTINE Prueba   (* ladder *)
END_ROUTINE
END_PROGRAM
